// /Chiller_2_Values
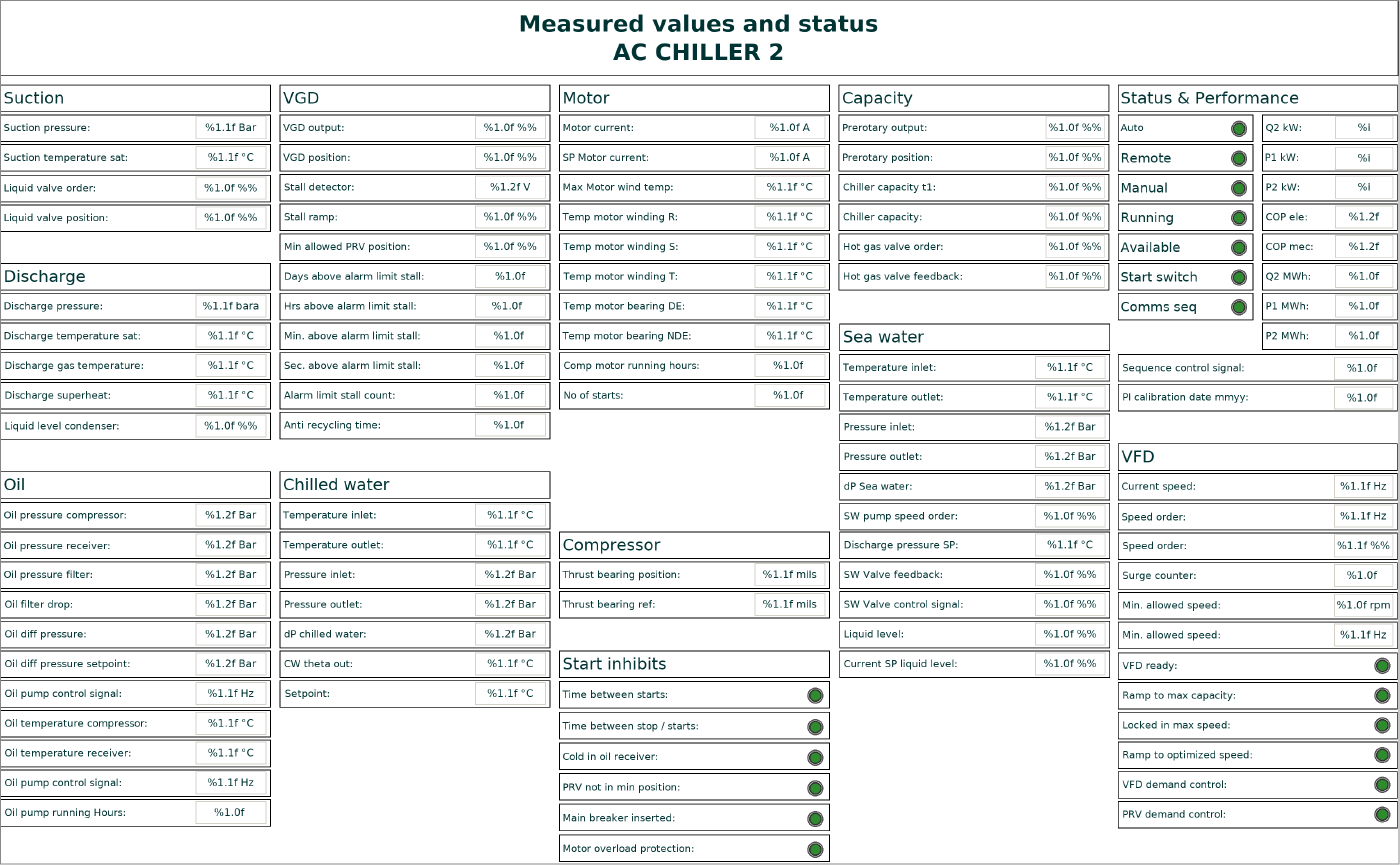
VISUALIZATION Chiller_2_Values  // 1553x960
    Rectangle (0,0 1551x84)
    Label (319,7 912x70), "Measured values and status AC CHILLER 2"
    Rectangle (0,94 300x30)
    Label (1,94 215x30), "Suction"
    Rectangle (0,127 300x30)
    Label (1,122 208x40), "Suction pressure:"
    Textfield (217,129 78x25), "%1.1f Bar", tooltip "Chiller_2.Press_suction_compr", text variable: Chiller_2.Press_suction_compr
        p4168582468: Chiller_2.Press_suction_compr
    Rectangle (0,160 300x30)
    Label (1,155 209x40), "Suction temperature sat:"
    Textfield (217,162 78x25), "%1.1f °C", tooltip "Chiller_2.Suction_saturated_temp", text variable: Chiller_2.Suction_saturated_temp
        p4168582468: Chiller_2.Suction_saturated_temp
    Rectangle (0,194 300x30)
    Label (1,189 211x40), "Liquid valve order:"
    Textfield (217,196 78x25), "%1.0f %%", tooltip "Chiller_2.Liquid_valve_output", text variable: Chiller_2.Liquid_valve_output
        p4168582468: Chiller_2.Liquid_valve_output
    Rectangle (0,227 300x30)
    Label (1,222 216x40), "Liquid valve position:"
    Textfield (217,229 78x25), "%1.0f %%", tooltip "Chiller_2.Feedback_liquid_valve", text variable: Chiller_2.Feedback_liquid_valve
        p4168582468: Chiller_2.Feedback_liquid_valve
    Rectangle (310,94 300x30)
    Label (311,94 194x30), "VGD"
    Rectangle (310,127 300x30)
    Label (311,122 209x40), "VGD output:"
    Textfield (527,129 78x25), "%1.0f %%", tooltip "Chiller_2.VGD_output", text variable: Chiller_2.VGD_output
        p4168582468: Chiller_2.VGD_output
    Rectangle (310,160 300x30)
    Label (311,155 204x40), "VGD position:"
    Textfield (527,162 78x25), "%1.0f %%", tooltip "Chiller_2.Feedback_VGD", text variable: Chiller_2.Feedback_VGD
        p4168582468: Chiller_2.Feedback_VGD
    Rectangle (310,193 300x30)
    Label (312,188 209x40), "Stall detector:"
    Textfield (527,195 78x25), "%1.2f V", tooltip "Chiller_2.Stall_detector", text variable: Chiller_2.Stall_detector
        p4168582468: Chiller_2.Stall_detector
    Rectangle (310,226 300x30)
    Label (312,221 178x40), "Stall ramp:"
    Textfield (527,228 78x25), "%1.0f %%", tooltip "Chiller_2.Stall_ramp", text variable: Chiller_2.Stall_ramp
        p4168582468: Chiller_2.Stall_ramp
    Rectangle (310,259 300x30)
    Label (312,254 216x40), "Min allowed PRV position:"
    Textfield (527,261 78x25), "%1.0f %%", tooltip "Chiller_2.Min_allowed_PRVposition", text variable: Chiller_2.Min_allowed_PRVposition
        p4168582468: Chiller_2.Min_allowed_PRVposition
    Rectangle (310,292 300x30)
    Label (312,287 216x40), "Days above alarm limit stall:"
    Textfield (527,294 78x25), "%1.0f", tooltip "Chiller_2.Days_above_stall_limit", text variable: Chiller_2.Days_above_stall_limit
        p4168582468: Chiller_2.Days_above_stall_limit
    Rectangle (310,325 300x30)
    Label (312,320 215x40), "Hrs above alarm limit stall:"
    Textfield (527,327 78x25), "%1.0f", tooltip "Chiller_2.Hrs_above_stall_limit", text variable: Chiller_2.Hrs_above_stall_limit
        p4168582468: Chiller_2.Hrs_above_stall_limit
    Rectangle (310,358 300x30)
    Label (312,353 218x40), "Min. above alarm limit stall:"
    Textfield (527,360 78x25), "%1.0f", tooltip "Chiller_2.Min_above_stall_limit", text variable: Chiller_2.Min_above_stall_limit
        p4168582468: Chiller_2.Min_above_stall_limit
    Rectangle (310,391 300x30)
    Label (312,386 214x40), "Sec. above alarm limit stall:"
    Textfield (527,393 78x25), "%1.0f", tooltip "Chiller_2.Sec_above_stall_limit", text variable: Chiller_2.Sec_above_stall_limit
        p4168582468: Chiller_2.Sec_above_stall_limit
    Rectangle (310,424 300x30)
    Label (312,419 216x40), "Alarm limit stall count:"
    Textfield (527,426 78x25), "%1.0f", tooltip "Chiller_2.Alarm_limit_stall_count", text variable: Chiller_2.Alarm_limit_stall_count
        p4168582468: Chiller_2.Alarm_limit_stall_count
    Rectangle (930,94 300x30)
    Label (931,94 162x30), "Capacity"
    Rectangle (930,127 300x30)
    Label (931,126 174x32), "Prerotary output:"
    Textfield (1160,129 65x25), "%1.0f %%", tooltip "Chiller_2.Prerotary_output", text variable: Chiller_2.Prerotary_output
        p4168582468: Chiller_2.Prerotary_output
    Rectangle (930,160 300x30)
    Label (931,159 173x32), "Prerotary position:"
    Textfield (1160,162 65x25), "%1.0f %%", tooltip "Chiller_2.Feedback_PRV", text variable: Chiller_2.Feedback_PRV
        p4168582468: Chiller_2.Feedback_PRV
    Rectangle (930,259 300x30)
    Label (932,258 177x32), "Hot gas valve order:"
    Textfield (1160,261 65x25), "%1.0f %%", tooltip "Chiller_2.Hot_gas_valve_output", text variable: Chiller_2.Hot_gas_valve_output
        p4168582468: Chiller_2.Hot_gas_valve_output
    Rectangle (930,292 300x30)
    Label (932,293 177x28), "Hot gas valve feedback:"
    Textfield (1160,294 65x25), "%1.0f %%", tooltip "Chiller_2.Feedback_HGV", text variable: Chiller_2.Feedback_HGV
        p4168582468: Chiller_2.Feedback_HGV
    Rectangle (0,292 300x30)
    Label (1,292 194x30), "Discharge"
    Rectangle (0,325 300x30)
    Label (1,320 213x40), "Discharge pressure:"
    Textfield (217,327 78x25), "%1.1f bara", tooltip "Chiller_2.Press_discharge_compr", text variable: Chiller_2.Press_discharge_compr
        p4168582468: Chiller_2.Press_discharge_compr
    Rectangle (0,358 300x30)
    Label (1,353 214x40), "Discharge temperature sat:"
    Textfield (217,360 78x25), "%1.1f °C", tooltip "Chiller_2.Discharge_saturated_temp", text variable: Chiller_2.Discharge_saturated_temp
        p4168582468: Chiller_2.Discharge_saturated_temp
    Rectangle (0,391 300x30)
    Label (2,386 213x40), "Discharge gas temperature:"
    Textfield (217,393 78x25), "%1.1f °C", tooltip "Chiller_2.Temp_discharge", text variable: Chiller_2.Temp_discharge
        p4168582468: Chiller_2.Temp_discharge
    Rectangle (0,458 300x30)
    Textfield (217,460 78x25), "%1.0f %%", tooltip "Chiller_2.Liquid_level_condenser", text variable: Chiller_2.Liquid_level_condenser
        p4168582468: Chiller_2.Liquid_level_condenser
    Rectangle (0,424 300x30)
    Label (2,419 212x40), "Discharge superheat:"
    Textfield (217,426 78x25), "%1.1f °C", tooltip "Chiller_2.Discharge_superheat", text variable: Chiller_2.Discharge_superheat
        p4168582468: Chiller_2.Discharge_superheat
    Label (2,453 210x40), "Liquid level condenser:"
    Rectangle (1240,127 150x30)
    Rectangle (1240,160 150x30)
    Rectangle (1240,193 150x30)
    Rectangle (1240,226 150x30)
    Rectangle (1240,259 150x30)
    Rectangle (1240,292 150x30)
    Rectangle (1240,325 150x30)
    Lamp1 (1363,133 23x20), tooltip "Chiller_2.Unit_auto", variable: Chiller_2.Unit_auto, style: Lamp-Lamp1-Green
    Label (1240,129 112x26), "Auto"
    Label (1240,165 105x21), "Remote"
    Lamp1 (1363,166 23x20), tooltip "Chiller_2.Unit_remote", variable: Chiller_2.Unit_remote, style: Lamp-Lamp1-Green
    Label (1240,198 105x21), "Manual"
    Lamp1 (1363,199 23x20), tooltip "Chiller_2.Unit_manual", variable: Chiller_2.Unit_manual, style: Lamp-Lamp1-Green
    Label (1240,231 105x21), "Running"
    Lamp1 (1363,232 23x20), tooltip "Chiller_2.Unit_running", variable: Chiller_2.Unit_running, style: Lamp-Lamp1-Green
    Label (1240,264 105x21), "Available"
    Lamp1 (1363,265 23x20), tooltip "Chiller_2.Unit_avabiable", variable: Chiller_2.Unit_available, style: Lamp-Lamp1-Green
    Label (1240,297 104x21), "Start switch"
    Lamp1 (1363,298 23x20), tooltip "Chiller_2.Unit_start_switch", variable: Chiller_2.Unit_start_switch, style: Lamp-Lamp1-Green
    Lamp1 (1363,331 23x20), tooltip "Sequence.A_Comms_Chiller_2", variable: not.Sequence.A_Comms_Chiller_2, style: Lamp-Lamp1-Green
    Label (1240,330 107x21), "Comms seq"
    Rectangle (930,193 300x30)
    Label (932,192 174x32), "Chiller capacity t1:"
    Textfield (1160,195 65x25), "%1.0f %%", tooltip "Chiller_2.Chiller_capacity_t1", text variable: Chiller_2.Chiller_capacity_t1
        p4168582468: Chiller_2.Chiller_capacity_t1
    Rectangle (620,94 300x30)
    Label (621,94 194x30), "Motor"
    Rectangle (620,127 300x30)
    Label (621,122 209x40), "Motor current:"
    Textfield (837,129 78x25), "%1.0f A", tooltip "Chiller_2.Motor_current", text variable: Chiller_2.Motor_current
        p4168582468: Chiller_2.Motor_current
    Rectangle (620,226 300x30)
    Label (621,221 210x40), "Temp motor winding R:"
    Textfield (837,228 78x25), "%1.1f °C", tooltip "Chiller_2.Temp_motor_wind_R", text variable: Chiller_2.Temp_motor_wind_R
        p4168582468: Chiller_2.Temp_motor_wind_R
    Rectangle (620,259 300x30)
    Label (622,254 204x40), "Temp motor winding S:"
    Textfield (837,261 78x25), "%1.1f °C", tooltip "Chiller_2.Temp_motor_wind_S", text variable: Chiller_2.Temp_motor_wind_S
        p4168582468: Chiller_2.Temp_motor_wind_S
    Rectangle (620,292 300x30)
    Label (622,287 206x40), "Temp motor winding T:"
    Textfield (837,294 78x25), "%1.1f °C", tooltip "Chiller_2.Temp_motor_wind_T", text variable: Chiller_2.Temp_motor_wind_T
        p4168582468: Chiller_2.Temp_motor_wind_T
    Rectangle (620,325 300x30)
    Label (622,320 216x40), "Temp motor bearing DE:"
    Textfield (837,327 78x25), "%1.1f °C", tooltip "Chiller_2.Temp_motor_bearing_DE", text variable: Chiller_2.Temp_motor_bearing_DE
        p4168582468: Chiller_2.Temp_motor_bearing_DE
    Rectangle (620,358 300x30)
    Label (621,353 218x40), "Temp motor bearing NDE:"
    Textfield (837,360 78x25), "%1.1f °C", tooltip "Chiller_2.Temp_motor_bearing_NDE", text variable: Chiller_2.Temp_motor_bearing_NDE
        p4168582468: Chiller_2.Temp_motor_bearing_NDE
    Rectangle (620,391 300x30)
    Label (622,386 214x40), "Comp motor running hours:"
    Textfield (837,393 78x25), "%1.0f", tooltip "Chiller_2.Running_hours_compressormotor", text variable: Chiller_2.Running_hours_compressormotor
        p4168582468: Chiller_2.Running_hours_compressormotor
    Rectangle (620,424 300x30)
    Label (622,419 207x40), "No of starts:"
    Textfield (837,426 78x25), "%1.0f", tooltip "Chiller_2.Number_of_starts", text variable: Chiller_2.Number_of_starts
        p4168582468: Chiller_2.Number_of_starts
    Rectangle (310,523 300x30)
    Label (311,523 194x30), "Chilled water"
    Rectangle (310,557 300x30)
    Label (311,552 204x40), "Temperature inlet:"
    Textfield (527,559 78x25), "%1.1f °C", tooltip "Chiller_2.Temp_chilled_medium_in", text variable: Chiller_2.Temp_chilled_medium_in
        p4168582468: Chiller_2.Temp_chilled_medium_in
    Rectangle (310,590 300x30)
    Label (311,585 209x40), "Temperature outlet:"
    Textfield (527,592 78x25), "%1.1f °C", tooltip "Chiller_2.Temp_chilled_medium_out", text variable: Chiller_2.Temp_chilled_medium_out
        p4168582468: Chiller_2.Temp_chilled_medium_out
    Rectangle (310,623 300x30)
    Label (312,618 206x40), "Pressure inlet:"
    Textfield (527,625 78x25), "%1.2f Bar", tooltip "Chiller_2.Press_chilled_medium_in", text variable: Chiller_2.Press_chilled_medium_in
        p4168582468: Chiller_2.Press_chilled_medium_in
    Rectangle (310,656 300x30)
    Label (312,651 208x40), "Pressure outlet:"
    Textfield (527,658 78x25), "%1.2f Bar", tooltip "Chiller_2.Press_chilled_medium_out", text variable: Chiller_2.Press_chilled_medium_out
        p4168582468: Chiller_2.Press_chilled_medium_out
    Rectangle (310,689 300x30)
    Label (312,684 207x40), "dP chilled water:"
    Textfield (527,691 78x25), "%1.2f Bar", tooltip "Chiller_2.dP_CW", text variable: Chiller_2.dP_CW
        p4168582468: Chiller_2.dP_CW
    Rectangle (310,722 300x30)
    Label (312,717 205x40), "CW theta out:"
    Textfield (527,724 78x25), "%1.1f °C", tooltip "Chiller_2.Theta_out", text variable: Chiller_2.Theta_out
        p4168582468: Chiller_2.Theta_out
    Rectangle (310,755 300x30)
    Label (313,750 205x40), "Setpoint:"
    Textfield (527,757 78x25), "%1.1f °C", tooltip "Chiller_2.SP_CW_controller", text variable: Chiller_2.SP_CW_controller
        p4168582468: Chiller_2.SP_CW_controller
    Rectangle (620,160 300x30)
    Label (621,155 209x40), "SP Motor current:"
    Textfield (837,162 78x25), "%1.0f A", tooltip "Chiller_2.SP_MC_controller", text variable: Chiller_2.SP_MC_controller
        p4168582468: Chiller_2.SP_MC_controller
    Rectangle (620,590 300x30)
    Label (621,590 194x30), "Compressor"
    Rectangle (620,623 300x30)
    Label (621,622 216x32), "Thrust bearing position:"
    Textfield (837,625 78x25), "%1.1f mils", tooltip "Chiller_2.Thrust_bearing_position", text variable: Chiller_2.Thrust_bearing_position
        p4168582468: Chiller_2.Thrust_bearing_position
    Rectangle (620,656 300x30)
    Label (621,655 216x32), "Thrust bearing ref:"
    Textfield (837,658 78x25), "%1.1f mils", tooltip "Chiller_2.Thrust_bearing_ref", text variable: Chiller_2.Thrust_bearing_ref
        p4168582468: Chiller_2.Thrust_bearing_ref
    Rectangle (310,457 300x30)
    Label (312,452 216x40), "Anti recycling time:"
    Textfield (527,459 78x25), "%1.0f", tooltip "Chiller_2.Anti_recycle_time", text variable: Chiller_2.Anti_recycle_time
        p4168582468: Chiller_2.Anti_recycle_time
    Rectangle (0,523 300x30)
    Label (1,523 194x30), "Oil"
    Rectangle (0,557 300x30)
    Label (1,552 211x40), "Oil pressure compressor:"
    Textfield (217,559 78x25), "%1.2f Bar", tooltip "Chiller_2.Press_oil_compr", text variable: Chiller_2.Press_oil_compr
        p4168582468: Chiller_2.Press_oil_compr
    Rectangle (0,590 300x30)
    Label (1,586 210x40), "Oil pressure receiver:"
    Textfield (217,592 78x25), "%1.2f Bar", tooltip "Chiller_2.Press_oil_receiver", text variable: Chiller_2.Press_oil_receiver
        p4168582468: Chiller_2.Press_oil_receiver
    Rectangle (0,656 300x30)
    Label (2,651 209x40), "Oil filter drop:"
    Textfield (217,658 78x25), "%1.2f Bar", tooltip "Chiller_2.Oil_Filter_Drop", text variable: Chiller_2.Oil_Filter_Drop
        p4168582468: Chiller_2.Oil_Filter_Drop
    Rectangle (0,689 300x30)
    Label (2,684 211x40), "Oil diff pressure:"
    Textfield (217,691 78x25), "%1.2f Bar", tooltip "Chiller_2.Oil_diff_pressure", text variable: Chiller_2.Oil_diff_pressure
        p4168582468: Chiller_2.Oil_diff_pressure
    Rectangle (0,788 300x30)
    Label (2,791 218x24), "Oil temperature compressor:"
    Textfield (217,790 78x25), "%1.1f °C", tooltip "Chiller_2.Temp_oil_inlet_compr", text variable: Chiller_2.Temp_oil_inlet_compr
        p4168582468: Chiller_2.Temp_oil_inlet_compr
    Rectangle (0,821 300x30)
    Label (2,816 210x40), "Oil temperature receiver:"
    Textfield (217,823 78x25), "%1.1f °C", tooltip "Chiller_2.Oil_temp_receiver", text variable: Chiller_2.Oil_temp_receiver
        p4168582468: Chiller_2.Oil_temp_receiver
    Rectangle (0,854 300x30)
    Label (2,849 212x40), "Oil pump control signal:"
    Textfield (217,856 78x25), "%1.1f Hz", tooltip "Chiller_2.Setpoint_conv_oil_pump", text variable: Chiller_2.Setpoint_conv_oil_pump
        p4168582468: Chiller_2.Setpoint_conv_oil_pump
    Rectangle (0,887 300x30)
    Label (2,882 206x40), "Oil pump running Hours:"
    Textfield (217,889 78x25), "%1.0f", tooltip "Chiller_2.Oil_pump_running_hours", text variable: Chiller_2.Oil_pump_running_hours
        p4168582468: Chiller_2.Oil_pump_running_hours
    Rectangle (0,623 300x30)
    Label (1,618 210x40), "Oil pressure filter:"
    Textfield (217,625 78x25), "%1.2f Bar", tooltip "Chiller_2.Oil_pressure_before_filter", text variable: Chiller_2.Oil_pressure_before_filter
        p4168582468: Chiller_2.Oil_pressure_before_filter
    Rectangle (0,722 300x30)
    Label (2,724 211x26), "Oil diff pressure setpoint:"
    Textfield (217,724 78x25), "%1.2f Bar", tooltip "Chiller_2.SP_oil_pressure", text variable: Chiller_2.SP_oil_pressure
        p4168582468: Chiller_2.SP_oil_pressure
    Rectangle (620,193 300x30)
    Label (621,188 210x40), "Max Motor wind temp:"
    Textfield (837,195 78x25), "%1.1f °C", tooltip "Chiller_2.Max_motor_wind_temp", text variable: Chiller_2.Max_motor_wind_temp
        p4168582468: Chiller_2.Max_motor_wind_temp
    Rectangle (931,359 300x30)
    Label (932,359 194x30), "Sea water"
    Rectangle (931,393 300x30)
    Label (932,388 211x40), "Temperature inlet:"
    Textfield (1148,395 78x25), "%1.1f °C", tooltip "Chiller_2.Temp_water_inlet_cond", text variable: Chiller_2.Temp_water_inlet_cond
        p4168582468: Chiller_2.Temp_water_inlet_cond
    Rectangle (931,459 300x30)
    Label (933,454 210x40), "Pressure inlet:"
    Textfield (1148,461 78x25), "%1.2f Bar", tooltip "Chiller_2.Press_water_cond_inlet", text variable: Chiller_2.Press_water_cond_inlet
        p4168582468: Chiller_2.Press_water_cond_inlet
    Rectangle (931,492 300x30)
    Label (933,487 210x40), "Pressure outlet:"
    Textfield (1148,494 78x25), "%1.2f Bar", tooltip "Chiller_2.Press_water_cond_out", text variable: Chiller_2.Press_water_cond_out
        p4168582468: Chiller_2.Press_water_cond_out
    Rectangle (931,525 300x30)
    Label (933,520 210x40), "dP Sea water:"
    Textfield (1148,527 78x25), "%1.2f Bar", tooltip "Chiller_2.dP_CW", text variable: Chiller_2.dP_SW
        p4168582468: Chiller_2.dP_SW
    Rectangle (931,558 300x30)
    Label (933,553 216x40), "SW pump speed order:"
    Textfield (1148,560 78x25), "%1.0f %%", tooltip "Chiller_2.SW_pump_speed_order", text variable: Chiller_2.SW_pump_speed_order
        p4168582468: Chiller_2.SW_pump_speed_order
    Rectangle (931,426 300x30)
    Label (932,421 211x40), "Temperature outlet:"
    Textfield (1148,428 78x25), "%1.1f °C", tooltip "Chiller_2.Temp_water_outlet_cond", text variable: Chiller_2.Temp_water_outlet_cond
        p4168582468: Chiller_2.Temp_water_outlet_cond
    Rectangle (931,590 300x30)
    Label (933,585 208x40), "Discharge pressure SP:"
    Textfield (1148,592 78x25), "%1.1f °C", tooltip "Chiller_2.SP_cond_press", text variable: Chiller_2.SP_cond_press
        p4168582468: Chiller_2.SP_cond_press
    Rectangle (931,623 300x30)
    Label (933,618 208x40), "SW Valve feedback:"
    Textfield (1148,625 78x25), "%1.0f %%", tooltip "Chiller_2.Feedback_seawater_valve_overboard", text variable: Chiller_2.Feedback_seawater_valve_overboard
        p4168582468: Chiller_2.Feedback_seawater_valve_overboard
    Rectangle (931,656 300x30)
    Label (933,651 208x40), "SW Valve control signal:"
    Textfield (1148,658 78x25), "%1.0f %%", tooltip "Chiller_2.Control_signal_SW_valve", text variable: Chiller_2.Order_SWW_overboard
        p4168582468: Chiller_2.Order_SWW_overboard
    Rectangle (931,689 300x30)
    Label (933,684 208x40), "Liquid level:"
    Textfield (1148,691 78x25), "%1.0f %%", tooltip "Chiller_2.Liquid_level_condenser", text variable: Chiller_2.Liquid_level_condenser
        p4168582468: Chiller_2.Liquid_level_condenser
    Rectangle (931,722 300x30)
    Label (933,717 208x40), "Current SP liquid level:"
    Textfield (1148,724 78x25), "%1.0f %%", tooltip "Chiller_2.SP_PID_Level", text variable: Chiller_2.SP_PID_Level
        p4168582468: Chiller_2.SP_PID_Level
    Rectangle (930,226 300x30)
    Label (932,225 174x32), "Chiller capacity:"
    Textfield (1160,228 65x25), "%1.0f %%", tooltip "Chiller_2.Chiller_capacity", text variable: Chiller_2.Chiller_capacity
        p4168582468: Chiller_2.Chiller_capacity
    Rectangle (1240,393 310x30)
    Label (1242,399 227x19), "Sequence control signal:"
    Textfield (1480,396 65x25), "%1.0f", tooltip "Chiller_2.Control_signal_unit_d", text variable: Chiller_2.Control_signal_unit_d
        p4168582468: Chiller_2.Control_signal_unit_d
    Rectangle (1240,426 310x30)
    Label (1242,429 227x24), "PI calibration date mmyy:"
    Textfield (1480,429 65x25), "%1.0f", tooltip "Chiller_2.Cal_date_MMYY", text variable: Chiller_2.Cal_date_MMYY
        p4168582468: Chiller_2.Cal_date_MMYY
    Rectangle (1400,226 150x30)
    Rectangle (1400,127 150x30)
    Rectangle (1400,193 150x30)
    Rectangle (1400,160 150x30)
    Rectangle (1400,292 150x30)
    Rectangle (1400,259 150x30)
    Rectangle (1400,358 150x30)
    Rectangle (1400,325 150x30)
    Label (1401,228 112x26), "COP ele:"
    Rectangle (1240,94 310x30)
    Label (1240,94 252x30), "Status & Performance"
    Label (1401,126 112x32), "Q2 kW:"
    Label (1401,194 112x28), "P2 kW:"
    Label (1400,159 112x32), "P1 kW:"
    Label (1401,293 112x28), "Q2 MWh:"
    Label (1401,261 112x26), "COP mec:"
    Label (1401,360 112x26), "P2 MWh:"
    Label (1401,327 112x26), "P1 MWh:"
    Textfield (1481,228 64x25), "%1.2f", tooltip "Chiller_2.COP_chiller_ele", text variable: Chiller_2.COP_chiller_ele
        p4168582468: Chiller_2.COP_chiller_ele
    Textfield (1481,129 64x25), "%i", tooltip "Chiller_2.Chiller_capacity_kW", text variable: Chiller_2.Chiller_capacity_kW
        p4168582468: Chiller_2.Chiller_capacity_kW
    Textfield (1481,195 64x25), "%i", tooltip "Chiller_2.P2_mot_1_kW", text variable: Chiller_2.P2_mot_1_kW
        p4168582468: Chiller_2.P2_mot_1_kW
    Textfield (1481,163 64x25), "%i", tooltip "Chiller_2.P1_motor_kW", text variable: Chiller_2.P1_motor_kW
        p4168582468: Chiller_2.P1_motor_kW
    Textfield (1481,294 64x25), "%1.0f", tooltip "Chiller_2.Q2_chillerMWh", text variable: Chiller_2.Q2_chillerMWh
        p4168582468: Chiller_2.Q2_chillerMWh
    Textfield (1481,261 64x25), "%1.2f", tooltip "Chiller_2.COP_chiller_mech", text variable: Chiller_2.COP_chiller_mech
        p4168582468: Chiller_2.COP_chiller_mech
    Textfield (1481,360 64x25), "%1.0f", tooltip "Chiller_2.Chiller_P2_MWh", text variable: Chiller_2.Chiller_P2_MWh
        p4168582468: Chiller_2.Chiller_P2_MWh
    Textfield (1481,327 64x25), "%1.0f", tooltip "Chiller_2.Chiller_P1_MWh", text variable: Chiller_2.Chiller_P1_MWh
        p4168582468: Chiller_2.Chiller_P1_MWh
    Rectangle (0,755 300x30)
    Label (2,757 211x26), "Oil pump control signal:"
    Textfield (217,757 78x25), "%1.1f Hz", tooltip "Chiller_2.Setpoint_conv_oil_pump", text variable: Chiller_2.Setpoint_conv_oil_pump
        p4168582468: Chiller_2.Setpoint_conv_oil_pump
    Rectangle (620,722 300x30)
    Label (621,722 194x30), "Start inhibits"
    Rectangle (620,756 300x30)
    Label (621,755 216x32), "Time between starts:"
    Rectangle (620,790 300x30)
    Label (621,790 216x32), "Time between stop / starts:"
    Rectangle (620,824 300x30)
    Label (621,824 216x32), "Cold in oil receiver:"
    Rectangle (620,858 300x30)
    Label (621,858 216x32), "PRV not in min position:"
    Rectangle (620,892 300x30)
    Label (621,892 216x32), "Main breaker inserted:"
    Lamp1 (893,762 23x20), variable: Chiller_2.Start_inhib_time_between_Start, style: Lamp-Lamp1-Green
    Lamp1 (893,797 23x20), variable: Chiller_2.Start_inhib_time_between_Stop_Start, style: Lamp-Lamp1-Green
    Lamp1 (893,831 23x20), variable: Chiller_2.Start_inhib_time_Oil_receiver_temp, style: Lamp-Lamp1-Green
    Lamp1 (893,865 23x20), variable: Chiller_2.Start_inhib_PRV_not_min, style: Lamp-Lamp1-Green
    Lamp1 (893,899 23x20), variable: not.Chiller_2.DO_9_0_Main_breaker_ready, style: Lamp-Lamp1-Green
    Rectangle (620,926 300x30)
    Label (621,926 216x32), "Motor overload protection:"
    Lamp1 (893,933 23x20), variable: not.Chiller_2.DI_0_6_Overload_protection, style: Lamp-Lamp1-Green
    Rectangle (1240,492 310x30)
    Rectangle (1240,525 310x30)
    Rectangle (1240,558 310x30)
    Rectangle (1240,591 310x30)
    Rectangle (1240,624 310x30)
    Rectangle (1240,657 310x30)
    Rectangle (1240,690 310x30)
    Rectangle (1240,724 310x30)
    Rectangle (1240,757 310x30)
    Rectangle (1240,790 310x30)
    Rectangle (1240,823 310x30)
    Rectangle (1240,856 310x30)
    Rectangle (1240,889 310x30)
    Label (1241,492 162x30), "VFD"
    Label (1241,524 173x32), "Current speed:"
    Textfield (1480,527 65x25), "%1.1f Hz", tooltip "Chiller_2.Speed_feedback_VFD", text variable: Chiller_2.Speed_feedback_VFD
        p4168582468: Chiller_2.Speed_feedback_VFD
    Label (1241,554 167x40), "Speed order:"
    Textfield (1480,560 65x25), "%1.1f Hz", tooltip "Chiller_2.Order_VFD_Hz", text variable: Chiller_2.Order_VFD_Hz
        p4168582468: Chiller_2.Order_VFD_Hz
    Label (1242,589 171x34), "Speed order:"
    Textfield (1480,593 65x25), "%1.1f %%", tooltip "Chiller_2.Opt_speed_VFD_perc", text variable: Chiller_2.Opt_speed_VFD_perc
        p4168582468: Chiller_2.Opt_speed_VFD_perc
    Label (1242,626 170x26), "Surge counter:"
    Textfield (1480,626 65x25), "%1.0f", tooltip "Chiller_2.Surge_counter_VFD", text variable: Chiller_2.Surge_counter_VFD
        p4168582468: Chiller_2.Surge_counter_VFD
    Label (1242,656 176x32), "Min. allowed speed:"
    Textfield (1480,659 65x25), "%1.0f rpm", tooltip "Chiller_2.VFD_min_allowed_speed", text variable: Chiller_2.VFD_min_allowed_speed
        p4168582468: Chiller_2.VFD_min_allowed_speed
    Label (1242,688 177x34), "Min. allowed speed:"
    Textfield (1480,692 65x25), "%1.1f Hz", tooltip "Chiller_2.VFD_min_allowed_frequence", text variable: Chiller_2.VFD_min_allowed_frequence
        p4168582468: Chiller_2.VFD_min_allowed_frequence
    Label (1242,722 177x34), "VFD ready:"
    Lamp1 (1522,729 23x20), tooltip "Chiller_2.VFD_ready", variable: Chiller_2.VFD_ready, style: Lamp-Lamp1-Green
    Label (1242,755 209x34), "Ramp to max capacity:"
    Lamp1 (1522,762 23x20), tooltip "Chiller_2.VFD_ramp_100_perc", variable: Chiller_2.VFD_ramp_100_perc, style: Lamp-Lamp1-Green
    Label (1242,788 209x34), "Locked in max speed:"
    Lamp1 (1522,795 23x20), tooltip "Chiller_2.VFD_locked_100_perc", variable: Chiller_2.VFD_locked_100_perc, style: Lamp-Lamp1-Green
    Label (1242,821 209x34), "Ramp to optimized speed:"
    Lamp1 (1522,828 23x20), tooltip "Chiller_2.VFD_ramp_d_PRVcontrol", variable: Chiller_2.VFD_ramp_d_PRVcontrol, style: Lamp-Lamp1-Green
    Label (1242,854 209x34), "VFD demand control:"
    Lamp1 (1522,861 23x20), tooltip "Chiller_2.VFD_control", variable: Chiller_2.VFD_control, style: Lamp-Lamp1-Green
    Label (1242,887 209x34), "PRV demand control:"
    Lamp1 (1522,894 23x20), tooltip "Chiller_2.PRV_control", variable: Chiller_2.PRV_control, style: Lamp-Lamp1-Green
END_VISUALIZATION

// /Chiller_2_VFD
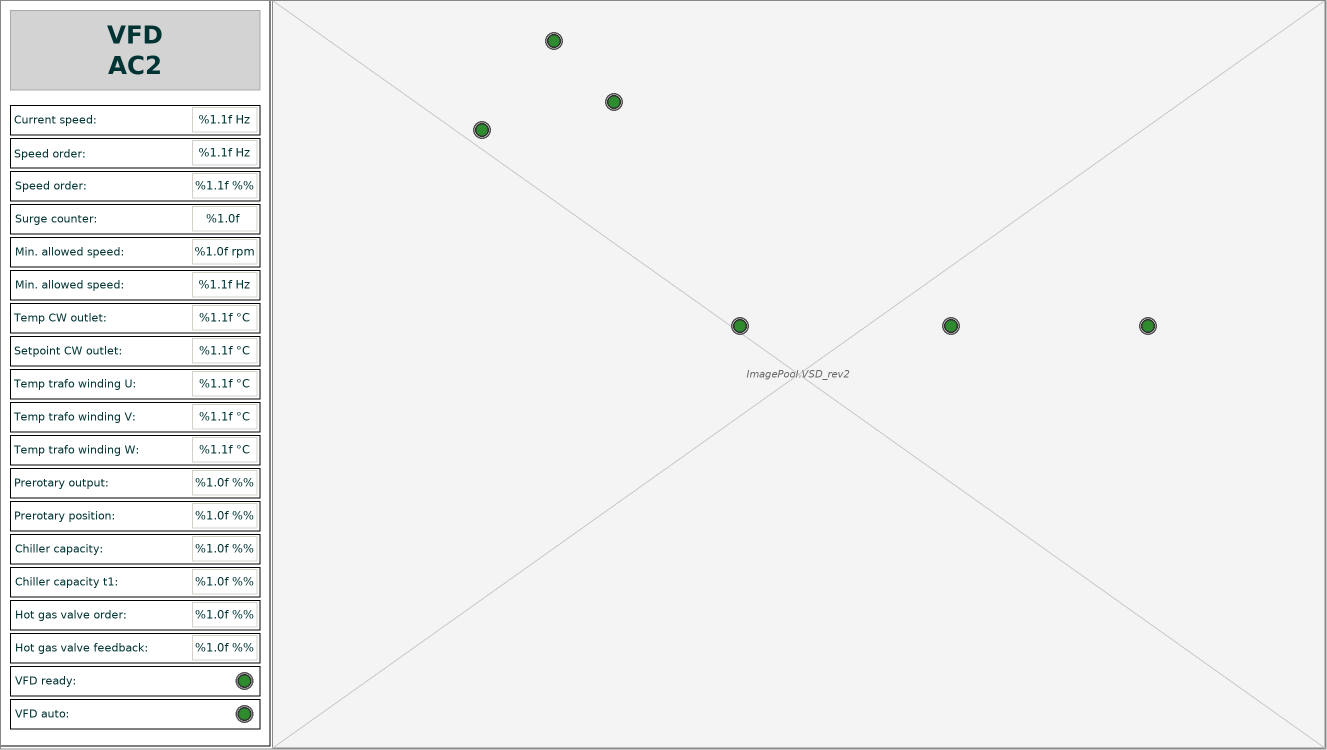
VISUALIZATION Chiller_2_VFD  // 1327x750
    Image (272,0 1053x748), image: ImagePool.VSD_rev2
    Rectangle (0,0 270x746)
    Lamp1 (469,120 26x20), variable: Chiller_2.VFD_ramp_100_perc, style: Lamp-Lamp1-Green
    Lamp1 (541,31 26x20), variable: Chiller_2.VFD_locked_100_perc, style: Lamp-Lamp1-Green
    Lamp1 (601,92 26x20), variable: Chiller_2.VFD_ramp_d_PRVcontrol, style: Lamp-Lamp1-Green
    Lamp1 (727,316 26x20), variable: Chiller_2.PRV_control, style: Lamp-Lamp1-Green
    Lamp1 (938,316 26x20), variable: Chiller_2.VFD_control, style: Lamp-Lamp1-Green
    Lamp1 (1135,316 26x20), variable: Chiller_2.PRV_control, style: Lamp-Lamp1-Green
    Textfield (10,10 250x80), "VFD AC2", text index: Sequence.Seq_cap_order_C3
    Rectangle (10,666 250x30)
    Label (12,664 177x34), "VFD ready:"
    Lamp1 (233,671 23x20), tooltip "Chiller_2.VFD_ready", variable: Chiller_2.VFD_ready, style: Lamp-Lamp1-Green
    Rectangle (10,699 250x30)
    Label (12,697 177x34), "VFD auto:"
    Lamp1 (233,704 23x20), tooltip "Chiller_2.VFD_man_auto", variable: Chiller_2.VFD_man_auto, style: Lamp-Lamp1-Green
    Rectangle (10,105 250x30)
    Label (11,104 173x32), "Current speed:"
    Textfield (192,107 65x25), "%1.1f Hz", tooltip "Chiller_2.Speed_feedback_VFD", text variable: Chiller_2.Speed_feedback_VFD
        p4168582468: Chiller_2.Speed_feedback_VFD
    Rectangle (10,138 250x30)
    Label (11,134 167x40), "Speed order:"
    Textfield (192,140 65x25), "%1.1f Hz", tooltip "Chiller_2.Order_VFD_Hz", text variable: Chiller_2.Order_VFD_Hz
        p4168582468: Chiller_2.Order_VFD_Hz
    Rectangle (10,171 250x30)
    Label (12,169 171x34), "Speed order:"
    Textfield (192,173 65x25), "%1.1f %%", tooltip "Chiller_2.Opt_speed_VFD_perc", text variable: Chiller_2.Opt_speed_VFD_perc
        p4168582468: Chiller_2.Opt_speed_VFD_perc
    Rectangle (10,204 250x30)
    Label (12,206 170x26), "Surge counter:"
    Textfield (192,206 65x25), "%1.0f", tooltip "Chiller_2.Surge_counter_VFD", text variable: Chiller_2.Surge_counter_VFD
        p4168582468: Chiller_2.Surge_counter_VFD
    Rectangle (10,237 250x30)
    Label (12,236 176x32), "Min. allowed speed:"
    Textfield (192,239 65x25), "%1.0f rpm", tooltip "Chiller_2.VFD_min_allowed_speed", text variable: Chiller_2.VFD_min_allowed_speed
        p4168582468: Chiller_2.VFD_min_allowed_speed
    Rectangle (10,270 250x30)
    Label (12,268 177x34), "Min. allowed speed:"
    Textfield (192,272 65x25), "%1.1f Hz", tooltip "Chiller_2.VFD_min_allowed_frequence", text variable: Chiller_2.VFD_min_allowed_frequence
        p4168582468: Chiller_2.VFD_min_allowed_frequence
    Rectangle (10,303 250x30)
    Label (11,305 169x26), "Temp CW outlet:"
    Textfield (192,305 65x25), "%1.1f °C", tooltip "Chiller_2.Temp_chilled_medium_out", text variable: Chiller_2.Temp_chilled_medium_out
        p4168582468: Chiller_2.Temp_chilled_medium_out
    Rectangle (10,336 250x30)
    Label (11,338 169x26), "Setpoint CW outlet:"
    Textfield (192,338 65x25), "%1.1f °C", tooltip "Chiller_2.SP_CW_controller", text variable: Chiller_2.SP_CW_controller
        p4168582468: Chiller_2.SP_CW_controller
    Rectangle (10,369 250x30)
    Label (11,371 169x26), "Temp trafo winding U:"
    Textfield (192,371 65x25), "%1.1f °C", tooltip "Chiller_2.Temp_motor_wind_R", text variable: Chiller_2.Temp_motor_wind_R
        p4168582468: Chiller_2.Temp_motor_wind_R
    Rectangle (10,402 250x30)
    Label (11,404 169x26), "Temp trafo winding V:"
    Textfield (192,404 65x25), "%1.1f °C", tooltip "Chiller_2.Temp_motor_wind_S", text variable: Chiller_2.Temp_motor_wind_S
        p4168582468: Chiller_2.Temp_motor_wind_S
    Rectangle (10,435 250x30)
    Label (11,437 169x26), "Temp trafo winding W:"
    Textfield (192,437 65x25), "%1.1f °C", tooltip "Chiller_2.Temp_motor_wind_T", text variable: Chiller_2.Temp_motor_wind_T
        p4168582468: Chiller_2.Temp_motor_wind_T
    Rectangle (10,468 250x30)
    Label (11,467 174x32), "Prerotary output:"
    Textfield (192,470 65x25), "%1.0f %%", tooltip "Chiller_2.Prerotary_output", text variable: Chiller_2.Prerotary_output
        p4168582468: Chiller_2.Prerotary_output
    Rectangle (10,501 250x30)
    Label (11,500 173x32), "Prerotary position:"
    Textfield (192,503 65x25), "%1.0f %%", tooltip "Chiller_2.Feedback_PRV", text variable: Chiller_2.Feedback_PRV
        p4168582468: Chiller_2.Feedback_PRV
    Rectangle (10,534 250x30)
    Label (12,533 174x32), "Chiller capacity:"
    Textfield (192,536 65x25), "%1.0f %%", tooltip "Chiller_2.Chiller_capacity", text variable: Chiller_2.Chiller_capacity
        p4168582468: Chiller_2.Chiller_capacity
    Rectangle (10,600 250x30)
    Label (12,599 177x32), "Hot gas valve order:"
    Textfield (192,602 65x25), "%1.0f %%", tooltip "Chiller_2.Hot_gas_valve_output", text variable: Chiller_2.Hot_gas_valve_output
        p4168582468: Chiller_2.Hot_gas_valve_output
    Rectangle (10,633 250x30)
    Label (12,634 177x28), "Hot gas valve feedback:"
    Textfield (192,635 65x25), "%1.0f %%", tooltip "Chiller_2.Feedback_HGV", text variable: Chiller_2.Feedback_HGV
        p4168582468: Chiller_2.Feedback_HGV
    Rectangle (10,567 250x30)
    Label (12,566 174x32), "Chiller capacity t1:"
    Textfield (192,569 65x25), "%1.0f %%", tooltip "Chiller_2.Chiller_capacity_t1", text variable: Chiller_2.Chiller_capacity_t1
        p4168582468: Chiller_2.Chiller_capacity_t1
    Rectangle (432,18 87x711), colour toggle: Chiller_2.VFD_ramp_100_perc
    Rectangle (518,18 65x711), colour toggle: Chiller_2.VFD_locked_100_perc
    Rectangle (583,18 57x711), colour toggle: Chiller_2.VFD_ramp_d_PRVcontrol
    Rectangle (641,18 199x711), colour toggle: Chiller_2.PRV_control
    Rectangle (1066,18 162x711), colour toggle: Chiller_2.PRV_control
    Rectangle (841,18 225x711), colour toggle: Chiller_2.VFD_control
END_VISUALIZATION

// /Chiller_3_Alarm
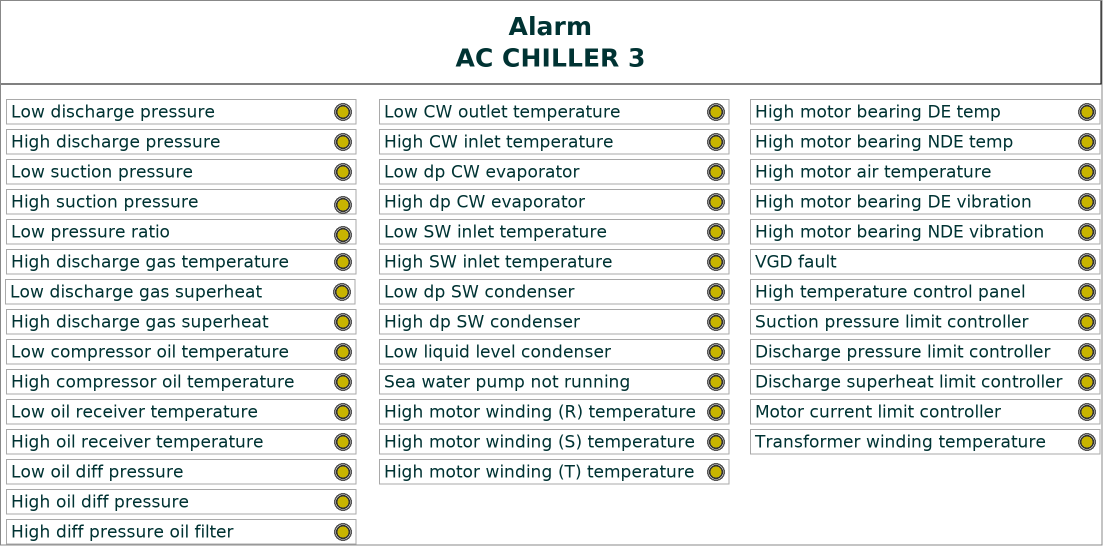
VISUALIZATION Chiller_3_Alarm  // 1103x546
    Rectangle (0,0 1101x84)
    Label (19,7 1063x70), "Alarm AC CHILLER 3"
    Rectangle (750,279 350x25)
    Label (752,281 316x21), "High temperature control panel"
    Lamp1 (1076,282 22x20), variable: Chiller_3.A_High_control_panel_temp, style: Lamp-Lamp1-Yellow
    Rectangle (750,309 350x25)
    Label (752,311 312x21), "Suction pressure limit controller"
    Lamp1 (1076,312 22x20), variable: Chiller_3.A_Suction_press_limit, style: Lamp-Lamp1-Yellow
    Rectangle (6,99 350x25)
    Label (8,101 318x21), "Low discharge pressure"
    Lamp1 (332,102 22x20), variable: Chiller_3.A_low_disch_press, style: Lamp-Lamp1-Yellow
    Rectangle (6,159 350x25)
    Label (8,161 319x21), "Low suction pressure"
    Lamp1 (332,162 22x20), variable: Chiller_3.A_Low_suction_pressure, style: Lamp-Lamp1-Yellow
    Rectangle (6,189 350x25)
    Label (8,191 322x21), "High suction pressure"
    Lamp1 (332,195 22x20), variable: Chiller_3.A_High_suction_pressure, style: Lamp-Lamp1-Yellow
    Rectangle (6,249 350x25)
    Label (8,251 317x21), "High discharge gas temperature"
    Lamp1 (332,252 22x20), variable: Chiller_3.A_High_discharge_temp, style: Lamp-Lamp1-Yellow
    Rectangle (379,399 350x25)
    Label (381,401 320x21), "High motor winding (R) temperature"
    Lamp1 (705,402 22x20), variable: Chiller_3.A_High_motor_wind_temp_R, style: Lamp-Lamp1-Yellow
    Rectangle (379,429 350x25)
    Label (381,431 319x21), "High motor winding (S) temperature"
    Lamp1 (705,432 22x20), variable: Chiller_3.A_High_motor_wind_temp_S, style: Lamp-Lamp1-Yellow
    Rectangle (6,369 350x25)
    Label (8,371 319x21), "High compressor oil temperature"
    Lamp1 (332,372 22x20), variable: Chiller_3.A_High_temp_oil_inlet_comp, style: Lamp-Lamp1-Yellow
    Rectangle (6,339 350x25)
    Label (8,341 322x21), "Low compressor oil temperature"
    Lamp1 (332,342 22x20), variable: Chiller_3.A_Low_temp_oil_inlet_comp, style: Lamp-Lamp1-Yellow
    Rectangle (6,429 350x25)
    Label (8,431 317x21), "High oil receiver temperature"
    Lamp1 (332,432 22x20), variable: Chiller_3.A_High_oil_temp_receiver, style: Lamp-Lamp1-Yellow
    Rectangle (6,399 350x25)
    Label (8,401 319x21), "Low oil receiver temperature"
    Lamp1 (332,402 22x20), variable: Chiller_3.A_Low_oil_temp_receiver, style: Lamp-Lamp1-Yellow
    Rectangle (6,459 350x25)
    Label (8,461 322x21), "Low oil diff pressure"
    Lamp1 (332,462 22x20), variable: Chiller_3.A_Low_oil_diff_pressure, style: Lamp-Lamp1-Yellow
    Rectangle (6,489 350x25)
    Label (8,491 317x21), "High oil diff pressure"
    Lamp1 (332,492 22x20), variable: Chiller_3.A_High_oil_diff_pressure, style: Lamp-Lamp1-Yellow
    Rectangle (6,309 350x25)
    Label (8,311 319x21), "High discharge gas superheat"
    Lamp1 (332,312 22x20), variable: Chiller_3.A_High_discharge_superheat, style: Lamp-Lamp1-Yellow
    Rectangle (5,279 350x25)
    Label (7,281 322x21), "Low discharge gas superheat"
    Lamp1 (331,282 22x20), variable: Chiller_3.A_Low_discharge_superheat, style: Lamp-Lamp1-Yellow
    Rectangle (379,219 350x25)
    Label (381,221 317x21), "Low SW inlet temperature"
    Lamp1 (705,222 22x20), variable: Chiller_3.A_Low_SW_inlet_temp, style: Lamp-Lamp1-Yellow
    Rectangle (379,129 350x25)
    Label (381,131 322x21), "High CW inlet temperature"
    Lamp1 (705,132 22x20), variable: Chiller_3.A_High_CW_inlet_temp, style: Lamp-Lamp1-Yellow
    Rectangle (379,99 350x25)
    Label (381,101 317x21), "Low CW outlet temperature"
    Lamp1 (705,102 22x20), variable: Chiller_3.A_Low_CW_outlet_temp, style: Lamp-Lamp1-Yellow
    Rectangle (6,519 350x25)
    Label (8,521 317x21), "High diff pressure oil filter"
    Lamp1 (332,522 22x20), variable: Chiller_3.A_High_oil_filter_diff_press, style: Lamp-Lamp1-Yellow
    Rectangle (379,459 350x25)
    Label (381,461 317x21), "High motor winding (T) temperature"
    Lamp1 (705,462 22x20), variable: Chiller_3.A_High_motor_wind_temp_T, style: Lamp-Lamp1-Yellow
    Rectangle (750,99 350x25)
    Label (752,101 317x21), "High motor bearing DE temp"
    Lamp1 (1076,102 22x20), variable: Chiller_3.A_High_comp_mo_DE_bear_temp, style: Lamp-Lamp1-Yellow
    Rectangle (750,129 350x25)
    Label (752,131 319x21), "High motor bearing NDE temp"
    Lamp1 (1076,132 22x20), variable: Chiller_3.A_High_comp_mo_NDE_bear_temp, style: Lamp-Lamp1-Yellow
    Rectangle (750,159 350x25)
    Label (752,161 322x21), "High motor air temperature"
    Lamp1 (1076,162 22x20), variable: Chiller_3.A_High_motor_air_temp, style: Lamp-Lamp1-Yellow
    Rectangle (750,189 350x25)
    Label (752,191 317x21), "High motor bearing DE vibration"
    Lamp1 (1076,192 22x20), variable: Chiller_3.A_High_comp_mo_DE_bear_vib, style: Lamp-Lamp1-Yellow
    Rectangle (750,219 350x25)
    Label (752,221 319x21), "High motor bearing NDE vibration"
    Lamp1 (1076,222 22x20), variable: Chiller_3.A_High_comp_mo_NDE_bear_vib, style: Lamp-Lamp1-Yellow
    Rectangle (379,189 350x25)
    Label (381,191 322x21), "High dp CW evaporator"
    Lamp1 (705,192 22x20), variable: Chiller_3.A_High_CW_dP, style: Lamp-Lamp1-Yellow
    Rectangle (379,159 350x25)
    Label (381,161 317x21), "Low dp CW evaporator"
    Lamp1 (705,162 22x20), variable: Chiller_3.A_Low_CW_dP, style: Lamp-Lamp1-Yellow
    Rectangle (379,309 350x25)
    Label (381,311 319x21), "High dp SW condenser"
    Lamp1 (705,312 22x20), variable: Chiller_3.A_High_SW_dP, style: Lamp-Lamp1-Yellow
    Rectangle (379,279 350x25)
    Label (381,281 322x21), "Low dp SW condenser"
    Lamp1 (705,282 22x20), variable: Chiller_3.A_Low_SW_dP, style: Lamp-Lamp1-Yellow
    Rectangle (750,249 350x25)
    Label (752,251 317x21), "VGD fault"
    Lamp1 (1076,252 22x20), variable: Chiller_3.A_VGD_Fault, style: Lamp-Lamp1-Yellow
    Rectangle (379,339 350x25)
    Label (381,341 317x21), "Low liquid level condenser"
    Lamp1 (705,342 22x20), variable: Chiller_3.A_Low_liquid_level, style: Lamp-Lamp1-Yellow
    Rectangle (6,129 350x25)
    Label (8,131 318x21), "High discharge pressure"
    Lamp1 (332,132 22x20), variable: Chiller_3.A_high_disch_press, style: Lamp-Lamp1-Yellow
    Rectangle (379,249 350x25)
    Label (381,251 314x21), "High SW inlet temperature"
    Lamp1 (705,252 22x20), variable: Chiller_3.A_High_SW_inlet_temp, style: Lamp-Lamp1-Yellow
    Rectangle (379,369 350x25)
    Label (381,371 314x21), "Sea water pump not running"
    Lamp1 (705,372 22x20), variable: Chiller_3.A_Seawater_pump_not_running, style: Lamp-Lamp1-Yellow
    Rectangle (750,339 350x25)
    Label (752,341 312x21), "Discharge pressure limit controller"
    Lamp1 (1076,342 22x20), variable: Chiller_3.A_Discharge_press_limit, style: Lamp-Lamp1-Yellow
    Rectangle (750,369 350x25)
    Label (752,371 312x21), "Discharge superheat limit controller"
    Lamp1 (1076,372 22x20), variable: Chiller_3.A_Discharge_superheat_limit, style: Lamp-Lamp1-Yellow
    Rectangle (750,399 350x25)
    Label (752,401 312x21), "Motor current limit controller"
    Lamp1 (1076,402 22x20), variable: Chiller_3.A_Motor_current_limit, style: Lamp-Lamp1-Yellow
    Rectangle (750,429 350x25)
    Label (752,431 312x21), "Transformer winding temperature"
    Lamp1 (1076,432 22x20), variable: Chiller_3.A_Transformer_winding_temp, style: Lamp-Lamp1-Yellow
    Rectangle (6,219 350x25)
    Label (8,221 322x21), "Low pressure ratio"
    Lamp1 (332,225 22x20), variable: Chiller_3.A_Low_press_ratio, style: Lamp-Lamp1-Yellow
END_VISUALIZATION

// /Chiller_3_Flow_Diagram
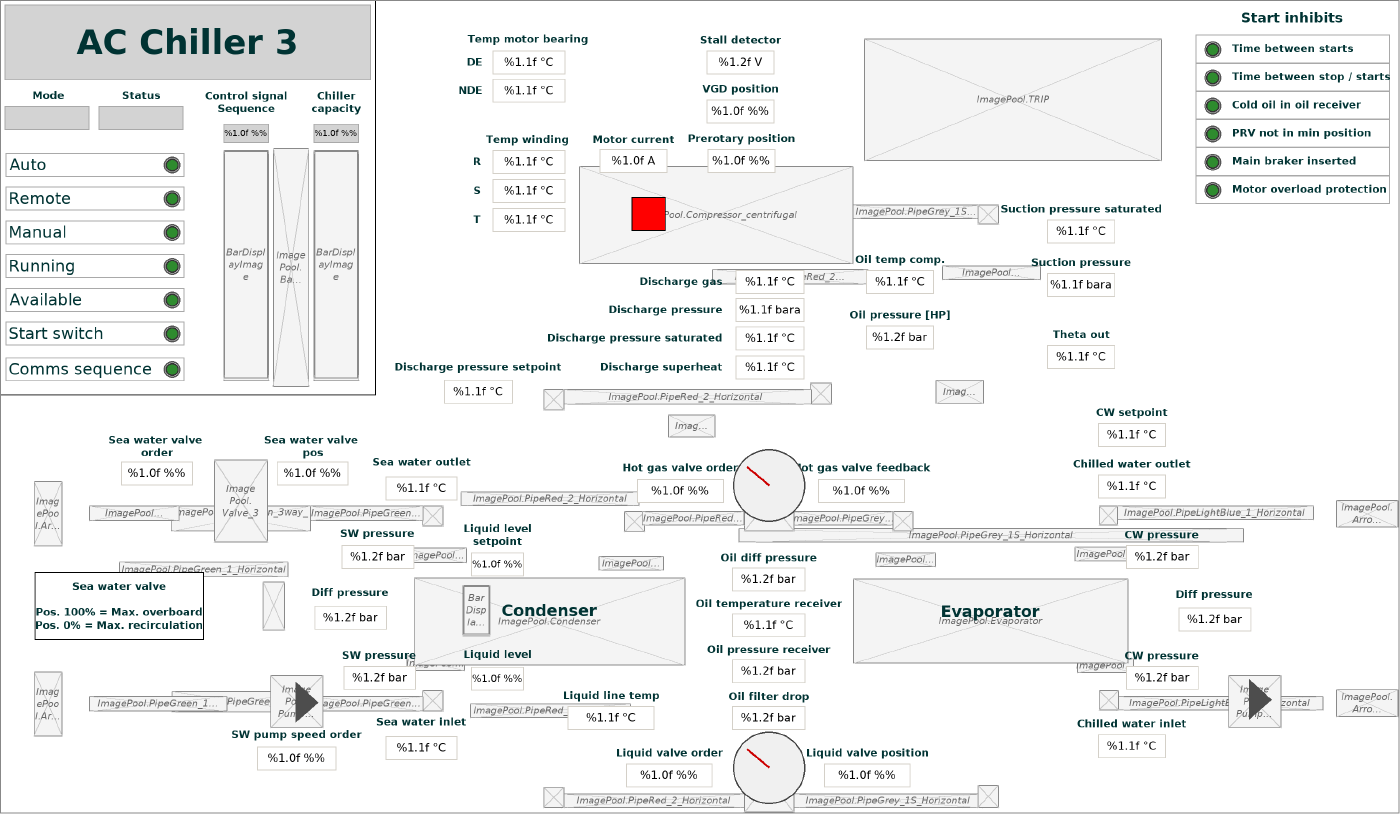
VISUALIZATION Chiller_3_Flow_Diagram  // 1492x868
    Rectangle (0,0 400x421)
    Textfield (238,132 48x20), "%1.0f %%", text variable: Sequence.Seq_cap_order_C3
        p4168582468: Sequence.Seq_cap_order_C3
    Image (1148,702 60x15), angle 270, image: ImagePool.PipeLightBlue_1_Horizontal
    Image (1145,583 67x15), angle 270, image: ImagePool.PipeLightBlue_1_Horizontal
    Image (908,218 137x15), image: ImagePool.PipeGrey_1S_Horizontal
    Image (845,846 202x15), image: ImagePool.PipeGrey_1S_Horizontal
    Image (933,589 64x15), angle 270, image: ImagePool.PipeGrey_1S_Horizontal
    Image (787,563 538x15), angle 270, image: ImagePool.PipeGrey_1S_Horizontal
    Image (843,545 110x15), image: ImagePool.PipeGrey_1S_Horizontal
    Image (638,593 69x15), angle 270, image: ImagePool.PipeRed_2_Horizontal
    Image (501,750 171x15), angle 270, image: ImagePool.PipeRed_2_Horizontal
    Label (218,94 89x30), "Control signal Sequence"
    Image (617,177 292x104), image: ImagePool.Compressor_centrifugal
    Image (759,287 166x16), angle 270, image: ImagePool.PipeRed_2_Horizontal
    Image (863,408 23x23), image: ImagePool.PipeRed_2_LU
    Image (596,415 269x16), image: ImagePool.PipeRed_2_Horizontal
    Image (909,617 293x90), image: ImagePool.Evaporator
    Image (431,584 66x16), angle 270, image: ImagePool.PipeGreen_1_Horizontal
    Image (450,539 22x22), image: ImagePool.PipeGreen_1_LD
    Image (329,539 122x16), image: ImagePool.PipeGreen_1_Horizontal
    Label (331,617 84x30), "Diff pressure"
    Textfield (335,646 77x25), "%1.2f bar", text variable: Chiller_3.dP_SW
        p4168582468: Chiller_3.dP_SW
    Image (127,599 180x16), angle 270, image: ImagePool.PipeGreen_1_Horizontal
    Image (183,737 147x22), image: ImagePool.PipeGreen_3way
    Image (433,699 62x16), angle 270, image: ImagePool.PipeGreen_1_Horizontal
    Image (450,736 22x22), image: ImagePool.PipeGreen_2_LU
    Image (329,742 122x16), image: ImagePool.PipeGreen_1_Horizontal
    Image (182,539 149x27), image: ImagePool.PipeGreen_3way_2
    Image (288,720 56x56), image: ImagePool.Pump_Large_3
    Polygon (315,746) (315,727) (339,749) (315,770) (315,762), colour toggle: Chiller_3.Sea_water_pump
    Image (36,513 30x69), angle 90, image: ImagePool.Arrow green down
    Image (36,716 30x69), angle 270, image: ImagePool.Arrow green down
    Image (579,415 22x22), image: ImagePool.PipeRed_1_RD
    Image (491,524 190x15), angle 270, image: ImagePool.PipeRed_2_Horizontal
    Label (360,554 84x30), "SW pressure"
    Textfield (364,581 77x25), "%1.2f bar", text variable: Chiller_3.Press_water_cond_out
        p4168582468: Chiller_3.Press_water_cond_out
    Image (95,539 96x16), image: ImagePool.PipeGreen_1_Horizontal
    Image (441,616 289x93), image: ImagePool.Condenser
    Image (598,846 197x15), image: ImagePool.PipeRed_2_Horizontal
    Image (579,839 22x22), image: ImagePool.PipeRed_2_RU
    Label (362,684 84x30), "SW pressure"
    Textfield (366,710 77x25), "%1.2f bar", text variable: Chiller_3.Press_water_cond_inlet
        p4168582468: Chiller_3.Press_water_cond_inlet
    Image (793,501 53x65), image: ImagePool.Valve_2
    Image (793,801 53x65), image: ImagePool.Valve_2
    Image (665,545 22x22), image: ImagePool.PipeRed_1_RD
    Image (684,545 109x15), image: ImagePool.PipeRed_2_Horizontal
    Image (951,545 22x21), image: ImagePool.PipeGrey_2_LD
    Image (1042,837 22x24), image: ImagePool.PipeGrey_3_LU
    Image (1042,218 22x21), image: ImagePool.PipeGrey_2_LD
    Image (1004,283 105x15), angle 270, image: ImagePool.PipeGrey_1S_Horizontal
    Label (521,636 129x30), "Condenser"
    Label (991,637 129x30), "Evaporator"
    Image (1189,539 211x15), image: ImagePool.PipeLightBlue_1_Horizontal
    Image (1171,539 20x21), image: ImagePool.PipeLightBlue_3_RD
    Image (1190,742 220x15), image: ImagePool.PipeLightBlue_1_Horizontal
    Image (1171,736 21x21), image: ImagePool.PipeLightBlue_3_RU
    Image (1424,533 66x29), angle 180, image: ImagePool.Arrow lightblue left
    Image (1424,735 66x29), image: ImagePool.Arrow lightblue left
    Image (1309,720 56x56), image: ImagePool.Pump_Large_3
    Polygon (1331,743) (1331,724) (1355,746) (1331,767) (1331,759), colour toggle: Chiller_3.CW_Flow_ind
    Image (280,620 23x52), image: ImagePool.Arrow green down
    Image (712,442 50x24), image: ImagePool.Arrow red left
    Image (997,405 51x25), angle 90, image: ImagePool.Arrow gray left
    Image (291,158 38x254), image: ImagePool.BarScale3
    Label (324,94 69x30), "Chiller capacity"
    Textfield (105,113 90x25), text list: 'TextList_PT', text index: Chiller_3.Unit_switch_status
    Textfield (5,113 90x25), text list: 'TextList_PT', text index: Chiller_3.Unit_start_switch
    Textfield (334,132 48x20), "%1.0f %%", text variable: Chiller_3.Chiller_capacity_t1
        p4168582468: Chiller_3.Chiller_capacity_t1
    Textfield (5,5 390x80), "AC Chiller 3"
    Textfield (525,160 77x25), "%1.1f °C", text variable: Chiller_3.Temp_motor_wind_R
        p4168582468: Chiller_3.Temp_motor_wind_R
    Label (496,160 25x25), "R"
    Textfield (525,191 77x25), "%1.1f °C", text variable: Chiller_3.Temp_motor_wind_S
        p4168582468: Chiller_3.Temp_motor_wind_S
    Label (496,191 25x25), "S"
    Textfield (525,222 77x25), "%1.1f °C", text variable: Chiller_3.Temp_motor_wind_T
        p4168582468: Chiller_3.Temp_motor_wind_T
    Label (496,222 25x25), "T"
    Textfield (679,511 92x25), "%1.0f %%", text variable: Chiller_3.Hot_gas_valve_output
        p4168582468: Chiller_3.Hot_gas_valve_output
    Label (664,484 122x30), "Hot gas valve order"
    Label (849,484 139x30), "Hot gas valve feedback"
    Textfield (872,511 92x25), "%1.0f %%", text variable: Chiller_3.Feedback_HGV
        p4168582468: Chiller_3.Feedback_HGV
    Meter360 (781,479 77x77), value: Chiller_3.Feedback_HGV, style: Meter-Meter360-Gray, scale format: %1.0f, scale 0..100
        p3451962224: ImagePool.Invisible
    Meter360 (781,780 77x77), value: Chiller_3.Feedback_liquid_valve, style: Meter-Meter360-Gray, scale format: %1.0f, scale 0..100
        p3451962224: ImagePool.Invisible
    Textfield (502,589 56x25), "%1.0f %%", text variable: Chiller_3.SP_PID_Level
        p4168582468: Chiller_3.SP_PID_Level
    Label (494,551 73x39), "Liquid level setpoint"
    Textfield (502,711 56x25), "%1.0f %%", text variable: Chiller_3.Liquid_level_condenser
        p4168582468: Chiller_3.Liquid_level_condenser
    Label (491,683 79x30), "Liquid level"
    Textfield (639,159 72x25), "%1.0f A", text variable: Chiller_3.Motor_current
        p4168582468: Chiller_3.Motor_current
    Label (634,138 83x22), "Motor current"
    Textfield (274,796 84x25), "%1.0f %%", text variable: Chiller_3.SW_pump_speed_order
        p4168582468: Chiller_3.SW_pump_speed_order
    Label (250,770 132x27), "SW pump speed order"
    Textfield (473,405 73x25), "%1.1f °C", tooltip "Chiller_3.SP_cond_press", text variable: Chiller_3.SP_cond_press
        p4168582468: Chiller_3.SP_cond_press
    Textfield (784,348 73x25), "%1.1f °C", text variable: Chiller_3.Discharge_saturated_temp
        p4168582468: Chiller_3.Discharge_saturated_temp
    Label (589,347 184x27), "Discharge pressure saturated"
    Label (425,378 169x27), "Discharge pressure setpoint"
    Textfield (411,785 76x25), "%1.1f °C", text variable: Chiller_3.Temp_water_inlet_cond
        p4168582468: Chiller_3.Temp_water_inlet_cond
    Label (399,755 100x30), "Sea water inlet"
    Textfield (411,508 76x25), "%1.1f °C", text variable: Chiller_3.Temp_water_outlet_cond
        p4168582468: Chiller_3.Temp_water_outlet_cond
    Label (397,478 105x30), "Sea water outlet"
    Label (500,27 126x30), "Temp motor bearing"
    Textfield (525,84 77x25), "%1.1f °C", text variable: Chiller_3.Temp_motor_bearing_NDE
        p4168582468: Chiller_3.Temp_motor_bearing_NDE
    Textfield (525,54 77x25), "%1.1f °C", text variable: Chiller_3.Temp_motor_bearing_DE
        p4168582468: Chiller_3.Temp_motor_bearing_DE
    Label (480,54 37x25), "DE"
    Label (480,84 37x25), "NDE"
    Label (678,287 95x27), "Discharge gas"
    Textfield (784,288 73x25), "%1.1f °C", text variable: Chiller_3.Temp_discharge
        p4168582468: Chiller_3.Temp_discharge
    Label (644,317 129x27), "Discharge pressure"
    Textfield (784,318 73x25), "%1.1f bara", text variable: Chiller_3.Press_discharge_compr
        p4168582468: Chiller_3.Press_discharge_compr
    Textfield (784,379 73x25), "%1.1f °C", text variable: Chiller_3.Discharge_superheat
        p4168582468: Chiller_3.Discharge_superheat
    Label (589,378 184x27), "Discharge superheat"
    Label (857,788 135x30), "Liquid valve position"
    Textfield (878,814 92x25), "%1.0f %%", text variable: Chiller_3.Feedback_liquid_valve
        p4168582468: Chiller_3.Feedback_liquid_valve
    Textfield (780,753 78x25), "%1.2f bar", text variable: Chiller_3.Oil_Filter_Drop
        p4168582468: Chiller_3.Oil_Filter_Drop
    Label (778,732 83x22), "Oil filter drop"
    Textfield (667,814 92x25), "%1.0f %%", text variable: Chiller_3.Liquid_valve_output
        p4168582468: Chiller_3.Liquid_valve_output
    Label (646,788 135x30), "Liquid valve order"
    Textfield (780,703 78x25), "%1.2f bar", text variable: Chiller_3.Press_oil_receiver
        p4168582468: Chiller_3.Press_oil_receiver
    Label (752,682 135x22), "Oil pressure receiver"
    Textfield (780,654 78x25), "%1.1f °C", text variable: Chiller_3.Oil_temp_receiver
        p4168582468: Chiller_3.Oil_temp_receiver
    Label (748,633 143x22), "Oil temperature receiver"
    Textfield (780,605 78x25), "%1.2f bar", text variable: Chiller_3.Oil_diff_pressure
        p4168582468: Chiller_3.Oil_diff_pressure
    Label (769,584 101x22), "Oil diff pressure"
    Label (736,136 109x24), "Prerotary position"
    Textfield (754,159 72x25), "%1.0f %%", text variable: Chiller_3.Feedback_PRV
        p4168582468: Chiller_3.Feedback_PRV
    Label (746,83 87x24), "VGD position"
    Textfield (753,106 72x25), "%1.0f %%", text variable: Chiller_3.Feedback_VGD
        p4168582468: Chiller_3.Feedback_VGD
    Label (746,31 87x24), "Stall detector"
    Textfield (753,54 72x25), "%1.2f V", text variable: Chiller_3.Stall_detector
        p4168582468: Chiller_3.Stall_detector
    Label (1067,211 171x24), "Suction pressure saturated"
    Textfield (1116,234 72x25), "%1.1f °C", text variable: Chiller_3.Suction_saturated_temp
        p4168582468: Chiller_3.Suction_saturated_temp
    Textfield (1116,291 72x25), "%1.1f bara", text variable: Chiller_3.Press_suction_compr
        p4168582468: Chiller_3.Press_suction_compr
    Label (1067,268 171x24), "Suction pressure"
    Textfield (1116,368 72x25), "%1.1f °C", text variable: Chiller_3.Theta_out
        p4168582468: Chiller_3.Theta_out
    Label (1111,345 83x24), "Theta out"
    Label (1196,557 84x27), "CW pressure"
    Textfield (1200,581 77x25), "%1.2f bar", text variable: Chiller_3.Press_chilled_medium_out
        p4168582468: Chiller_3.Press_chilled_medium_out
    Textfield (1200,710 77x25), "%1.2f bar", text variable: Chiller_3.Press_chilled_medium_in
        p4168582468: Chiller_3.Press_chilled_medium_in
    Label (1196,686 84x27), "CW pressure"
    Textfield (1170,506 72x25), "%1.1f °C", text variable: Chiller_3.Temp_chilled_medium_out
        p4168582468: Chiller_3.Temp_chilled_medium_out
    Label (1146,483 121x24), "Chilled water outlet"
    Label (1146,428 121x24), "CW setpoint"
    Textfield (1170,451 72x25), "%1.1f °C", text variable: Chiller_3.SP_CW_controller
        p4168582468: Chiller_3.SP_CW_controller
    Label (1252,619 84x30), "Diff pressure"
    Textfield (1256,648 77x25), "%1.2f bar", text variable: Chiller_3.dP_CW
        p4168582468: Chiller_3.dP_CW
    Textfield (1170,783 72x25), "%1.1f °C", text variable: Chiller_3.Temp_chilled_medium_in
        p4168582468: Chiller_3.Temp_chilled_medium_in
    Label (1146,760 121x24), "Chilled water inlet"
    Group (6,271 190x25)
        Rectangle (0,0 190x25)
        Label (0,2 105x21), "Running"
        Lamp1 (166,3 23x20), variable: Chiller_3.Unit_running, style: Lamp-Lamp1-Green
    Group (6,163 190x25)
        Rectangle (0,0 190x25)
        Label (1,2 105x21), "Auto"
        Lamp1 (166,3 23x20), variable: Chiller_3.Unit_auto, style: Lamp-Lamp1-Green
    Group (6,199 190x25)
        Rectangle (0,0 190x25)
        Label (0,2 105x21), "Remote"
        Lamp1 (166,3 23x20), variable: Chiller_3.Unit_remote, style: Lamp-Lamp1-Green
    Group (6,235 190x25)
        Rectangle (0,0 190x25)
        Label (0,2 105x21), "Manual"
        Lamp1 (166,3 23x20), variable: Chiller_3.Unit_manual, style: Lamp-Lamp1-Green
    Group (6,307 190x25)
        Rectangle (0,0 190x25)
        Label (1,2 105x21), "Available"
        Lamp1 (166,3 23x20), variable: Chiller_3.Unit_available, style: Lamp-Lamp1-Green
    Group (6,343 190x25)
        Rectangle (0,0 190x25)
        Label (0,2 130x21), "Start switch"
        Lamp1 (166,3 23x20), variable: Chiller_3.Unit_start_switch, style: Lamp-Lamp1-Green
    Group (6,381 190x25)
        Rectangle (0,0 190x25)
        Label (0,2 160x21), "Comms sequence"
        Lamp1 (166,3 23x20), variable: not.Sequence.A_Comms_Chiller_3, style: Lamp-Lamp1-Green
    Label (912,265 95x24), "Oil temp comp."
    Textfield (923,288 72x25), "%1.1f °C", text variable: Chiller_3.Temp_oil_inlet_compr
        p4168582468: Chiller_3.Temp_oil_inlet_compr
    Label (902,324 115x24), "Oil pressure [HP]"
    Textfield (923,347 72x25), "%1.2f bar", text variable: Chiller_3.Press_oil_compr
        p4168582468: Chiller_3.Press_oil_compr
    Image (921,41 317x130), invisible if: Chiller_3.Unit_alarm, image: ImagePool.ALARM
    Image (921,41 317x130), invisible if: Chiller_3.Unit_trip, image: ImagePool.TRIP
    Label (7,87 89x30), "Mode"
    Label (106,87 89x30), "Status"
    Rectangle (334,160 48x246)
    Image (238,160 48x246), image: ImagePool.CapBarTranparant
    BarDisplayImage (239,161 46x242), value: Sequence.Seq_cap_order_C3, style: BarDisplayImage-Gray, scale format: %.0f, scale 0..100
        p3451962224: ImagePool.Invisible
    Rectangle (673,210 36x36), colour toggle: Chiller_3.Unit_running
    Rectangle (673,210 36x36), colour toggle: Chiller_3.Unit_alarm
    Rectangle (673,210 36x36), colour toggle: Chiller_3.Unit_trip
    Image (334,160 48x246), image: ImagePool.CapBarTranparant
    BarDisplayImage (335,161 46x242), value: Chiller_3.Chiller_capacity_t1, style: BarDisplayImage-Gray, scale format: %.0f, scale 0..100
        p3451962224: ImagePool.Invisible
    Rectangle (493,624 28x52)
    Image (493,624 29x54), image: ImagePool.CapBarTranparant
    BarDisplayImage (494,625 27x51), value: Chiller_3.Liquid_level_condenser, style: BarDisplayImage-Gray, scale format: %.0f, scale 0..100
        p3451962224: ImagePool.Invisible
    Image (95,742 147x16), image: ImagePool.PipeGreen_1_Horizontal
    Textfield (605,753 92x25), "%1.1f °C", text variable: Chiller_3.Liquid_line_temp
        p4168582468: Chiller_3.Liquid_line_temp
    Label (595,727 113x30), "Liquid line temp"
    Image (228,490 57x88), image: ImagePool.Valve_3
    Label (115,461 105x30), "Sea water valve order"
    Textfield (129,492 76x25), "%1.0f %%", text variable: Chiller_3.Order_SWW_overboard
        p4168582468: Chiller_3.Order_SWW_overboard
    Label (281,461 105x30), "Sea water valve pos"
    Textfield (295,492 76x25), "%1.0f %%", text variable: Chiller_3.Feedback_seawater_valve_overboard
        p4168582468: Chiller_3.Feedback_seawater_valve_overboard
    Group (37,610 180x72)
        Rectangle (0,0 180x72)
        Label (0,0 180x72), "Sea water valve Pos. 100% = Max. overboard Pos. 0% = Max. recirculation"
    Label (511,138 103x22), "Temp winding"
    Rectangle (1274,37 207x30)
    Label (1310,38 142x28), "Time between starts"
    Lamp1 (1281,43 23x20), variable: Chiller_3.Start_inhib_time_between_Start, style: Lamp-Lamp1-Green
    Rectangle (1274,67 207x30)
    Label (1310,68 162x28), "Time between stop / starts"
    Lamp1 (1281,73 23x20), variable: Chiller_3.Start_inhib_time_between_Stop_Start, style: Lamp-Lamp1-Green
    Label (1307,7 140x24), "Start inhibits"
    Rectangle (1274,97 207x30)
    Label (1310,98 162x28), "Cold oil in oil receiver"
    Lamp1 (1281,103 23x20), variable: Chiller_3.Start_inhib_time_Oil_receiver_temp, style: Lamp-Lamp1-Green
    Rectangle (1274,127 207x30)
    Label (1310,128 162x28), "PRV not in min position"
    Lamp1 (1281,133 23x20), variable: Chiller_3.Start_inhib_PRV_not_min, style: Lamp-Lamp1-Green
    Rectangle (1274,157 207x30)
    Label (1310,158 162x28), "Main braker inserted"
    Lamp1 (1281,163 23x20), variable: not.Chiller_3.DO_9_0_Main_breaker_ready, style: Lamp-Lamp1-Green
    Rectangle (1274,187 207x30)
    Label (1310,188 162x28), "Motor overload protection"
    Lamp1 (1281,193 23x20), variable: not.Chiller_3.DI_0_6_Overload_protection, style: Lamp-Lamp1-Green
END_VISUALIZATION

// /Chiller_3_Oil
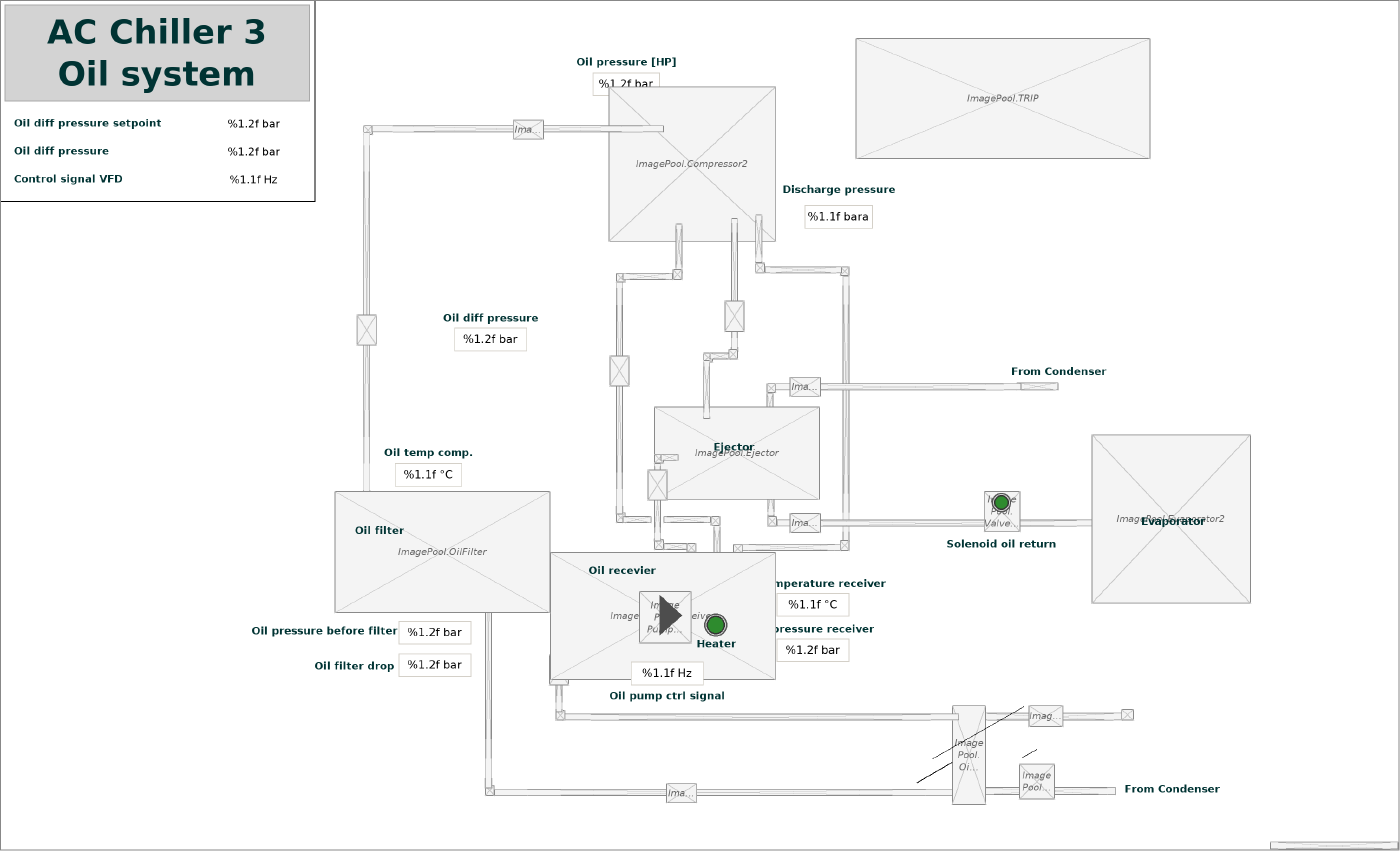
VISUALIZATION Chiller_3_Oil  // 1507x917
    Image (1094,412 45x8), angle 180, image: ImagePool.PipeBlack_1S_H_Faded
    Rectangle (0,0 339x217)
    Image (1367,907 138x8), angle 270, image: ImagePool.PipeGrey_1S_Horizontal
    Image (1053,768 155x8), image: ImagePool.PipeGrey_1S_Horizontal
    Image (1207,764 13x12), image: ImagePool.PipeGrey_3_LU
    Textfield (5,5 328x104), "AC Chiller 3 Oil system"
    Label (1066,387 128x27), "From Condenser"
    Label (838,191 129x27), "Discharge pressure"
    Textfield (866,221 73x25), "%1.1f bara", text variable: Chiller_3.Press_discharge_compr
        p4168582468: Chiller_3.Press_discharge_compr
    Label (1007,573 142x27), "Solenoid oil return"
    Textfield (429,704 78x25), "%1.2f bar", text variable: Chiller_3.Oil_Filter_Drop
        p4168582468: Chiller_3.Oil_Filter_Drop
    Label (340,707 83x22), "Oil filter drop"
    Textfield (836,688 78x25), "%1.2f bar", text variable: Chiller_3.Press_oil_receiver
        p4168582468: Chiller_3.Press_oil_receiver
    Label (808,667 135x22), "Oil pressure receiver"
    Textfield (836,639 78x25), "%1.1f °C", text variable: Chiller_3.Oil_temp_receiver
        p4168582468: Chiller_3.Oil_temp_receiver
    Label (804,618 143x22), "Oil temperature receiver"
    Textfield (489,353 78x25), "%1.2f bar", text variable: Chiller_3.Oil_diff_pressure
        p4168582468: Chiller_3.Oil_diff_pressure
    Label (478,332 101x22), "Oil diff pressure"
    Label (414,476 95x24), "Oil temp comp."
    Textfield (425,499 72x25), "%1.1f °C", text variable: Chiller_3.Temp_oil_inlet_compr
        p4168582468: Chiller_3.Temp_oil_inlet_compr
    Label (617,55 115x24), "Oil pressure [HP]"
    Textfield (638,78 72x25), "%1.2f bar", text variable: Chiller_3.Press_oil_compr
        p4168582468: Chiller_3.Press_oil_compr
    Image (921,41 317x130), invisible if: Chiller_3.Unit_alarm, image: ImagePool.ALARM
    Image (921,41 317x130), invisible if: Chiller_3.Unit_trip, image: ImagePool.TRIP
    Textfield (238,122 70x23), "%1.2f bar", text variable: Chiller_3.SP_oil_pressure
    Label (12,118 193x30), "Oil diff pressure setpoint"
    Textfield (238,152 70x23), "%1.2f bar", text variable: Chiller_3.Oil_diff_pressure
    Label (12,148 193x30), "Oil diff pressure"
    Textfield (238,182 70x23), "%1.1f Hz", text variable: Chiller_3.Setpoint_conv_oil_pump
    Label (12,178 131x30), "Control signal VFD"
    Label (651,739 135x22), "Oil pump ctrl signal"
    Textfield (429,669 78x25), "%1.2f bar", text variable: Chiller_3.Oil_pressure_before_filter
        p4168582468: Chiller_3.Oil_pressure_before_filter
    Label (276,669 147x22), "Oil pressure before filter"
    Label (1210,837 106x27), "From Condenser"
    Image (655,93 180x167), image: ImagePool.Compressor2
    Image (1051,848 150x8), angle 180, image: ImagePool.PipeBlack_1S_H_Faded
    Image (798,586 108x7), image: ImagePool.PipeBlack_1_Horizontal
    Image (907,297 7x286), image: ImagePool.PipeBlack_1_Vertical
    Image (391,135 10x10), image: ImagePool.PipeBlack_1_RD
    Image (522,846 10x11), image: ImagePool.PipeBlack_1_RU
    Image (1107,760 37x23), image: ImagePool.Arrow gray right
    Image (836,560 348x7), image: ImagePool.PipeBlack_1_Horizontal
    Image (1175,468 171x182), image: ImagePool.Evaporator2
    Image (826,512 7x44), image: ImagePool.PipeBlack_1_Vertical
    Image (826,556 10x11), image: ImagePool.PipeBlack_1_RU
    Image (789,596 7x28), image: ImagePool.PipeBlack_1_Vertical
    Image (789,586 10x10), image: ImagePool.PipeBlack_1_RD
    Image (904,582 10x11), image: ImagePool.PipeBlack_1_LU
    Image (850,553 33x21), image: ImagePool.Arrow black left
    Image (904,287 10x10), image: ImagePool.PipeBlack_1_LD
    Image (823,287 83x7), image: ImagePool.PipeBlack_1_Horizontal
    Image (813,283 10x11), image: ImagePool.PipeBlack_1_RU
    Image (813,231 7x52), image: ImagePool.PipeBlack_1_Vertical
    Image (825,413 10x10), image: ImagePool.PipeBlack_1_RD
    Image (834,413 265x7), image: ImagePool.PipeBlack_1_Horizontal
    Image (825,423 7x28), image: ImagePool.PipeBlack_1_Vertical
    Image (704,438 178x100), image: ImagePool.Ejector
    Image (850,406 33x21), image: ImagePool.Arrow black left
    Image (532,850 500x7), image: ImagePool.PipeBlack_1_Horizontal
    Image (1025,760 36x107), image: ImagePool.OilHeatExchanger
    Image (605,769 427x7), image: ImagePool.PipeBlack_1_Horizontal
    Image (598,765 10x11), image: ImagePool.PipeBlack_1_RU
    Image (598,670 7x97), image: ImagePool.PipeBlack_1_Vertical
    Image (598,660 10x10), image: ImagePool.PipeBlack_1_RD
    Image (605,660 19x7), image: ImagePool.PipeBlack_1_Horizontal
    Image (591,705 21x33), image: ImagePool.Arrow black down
    Image (717,844 33x21), image: ImagePool.Arrow black left
    Image (768,566 7x50), image: ImagePool.PipeBlack_1_Vertical
    Image (765,556 10x10), image: ImagePool.PipeBlack_1_LD
    Image (714,556 51x7), image: ImagePool.PipeBlack_1_Horizontal
    Image (704,581 10x11), image: ImagePool.PipeBlack_1_RU
    Image (704,499 7x84), image: ImagePool.PipeBlack_1_Vertical
    Image (704,489 10x10), image: ImagePool.PipeBlack_1_RD
    Image (711,489 19x7), image: ImagePool.PipeBlack_1_Horizontal
    Image (697,506 21x33), image: ImagePool.Arrow black down
    Image (714,585 28x7), image: ImagePool.PipeBlack_1_Horizontal
    Image (739,585 10x10), image: ImagePool.PipeBlack_1_LD
    Image (742,595 7x21), image: ImagePool.PipeBlack_1_Vertical
    Image (592,595 243x137), image: ImagePool.OilReceiver
    Image (400,135 314x7), image: ImagePool.PipeBlack_1_Horizontal
    Label (630,604 80x22), "Oil recevier"
    Image (522,553 7x296), image: ImagePool.PipeBlack_1_Vertical
    Image (519,544 10x10), image: ImagePool.PipeBlack_1_LD
    Image (400,544 120x7), image: ImagePool.PipeBlack_1_Horizontal
    Image (391,540 10x11), image: ImagePool.PipeBlack_1_RU
    Image (391,142 7x400), image: ImagePool.PipeBlack_1_Vertical
    Image (663,552 10x11), image: ImagePool.PipeBlack_1_RU
    Image (663,301 7x253), image: ImagePool.PipeBlack_1_Vertical
    Image (663,294 10x10), image: ImagePool.PipeBlack_1_RD
    Image (670,294 54x7), image: ImagePool.PipeBlack_1_Horizontal
    Image (656,383 21x33), image: ImagePool.Arrow black down
    Image (670,556 31x7), image: ImagePool.PipeBlack_1_Horizontal
    Image (727,241 7x53), image: ImagePool.PipeBlack_1_Vertical
    Image (724,290 10x11), image: ImagePool.PipeBlack_1_LU
    Image (757,380 10x10), image: ImagePool.PipeBlack_1_RD
    Image (764,380 22x7), image: ImagePool.PipeBlack_1_Horizontal
    Image (787,235 7x144), image: ImagePool.PipeBlack_1_Vertical
    Image (784,376 10x11), image: ImagePool.PipeBlack_1_LU
    Image (757,388 7x63), image: ImagePool.PipeBlack_1_Vertical
    Image (780,324 21x33), image: ImagePool.Arrow black down
    Label (750,471 80x22), "Ejector"
    Label (1223,551 80x22), "Evaporator"
    Image (384,339 21x33), image: ImagePool.Arrow black up
    Image (552,129 33x21), image: ImagePool.Arrow black right
    Image (360,529 232x131), image: ImagePool.OilFilter
    Label (379,561 59x22), "Oil filter"
    Line (987,843) (1025,821)
    Line (1100,816) (1116,807)
    Line (1004,817) (1102,761)
    Image (1097,823 38x38), image: ImagePool.RegValve
    Image (688,637 56x56), image: ImagePool.Pump_Large_3
    Polygon (710,660) (710,641) (734,663) (710,684) (710,676), colour toggle: Chiller_3.Comp_oil_pump
    Lamp1 (756,656 29x35), variable: Chiller_3.DO_0_6_Oil_heater, style: Lamp-Lamp1-Green
    Label (744,683 55x22), "Heater"
    Image (1059,529 39x44), image: ImagePool.Valve_2
    Lamp1 (1066,529 24x25), variable: Chiller_3.DO_0_4_Solenoid_valve_oil, style: Lamp-Lamp1-Green
    Textfield (679,713 78x25), "%1.1f Hz", text variable: Chiller_3.Setpoint_conv_oil_pump
END_VISUALIZATION

// /Homepage
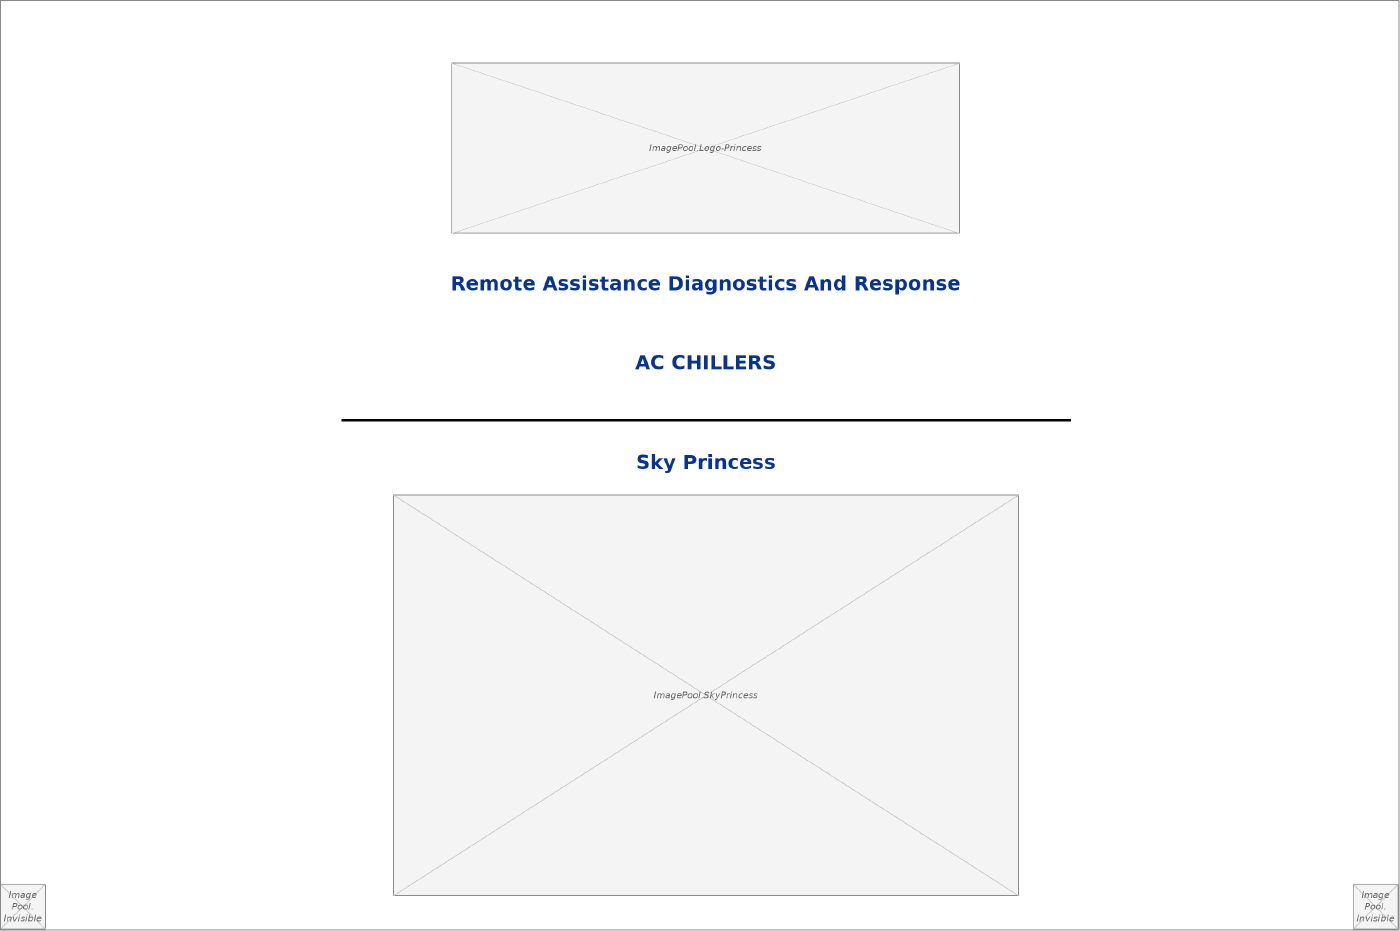
VISUALIZATION Homepage  // 1542x1026
    Label (490,287 575x51), "Remote Assistance Diagnostics And Response"
    Label (597,484 361x51), "Sky Princess"
    Rectangle (376,462 803x2)
    Label (597,374 361x51), "AC CHILLERS"
    Image (0,974 50x50), image: ImagePool.Invisible
    Image (1490,974 50x50), image: ImagePool.Invisible
    Image (433,545 689x442), image: ImagePool.SkyPrincess
    Image (497,69 560x188), image: ImagePool.Logo-Princess
END_VISUALIZATION

(* text list Chiller_trendvalues (id | default)
  0 | Clear values
  1 | Chiller Capacity t1
  2 | Control Signal SW Valve
  3 | dP CW
  4 | dP SW
  5 | Feedback Hot Gas Valve
  6 | Feedback Liquid Valve
  7 | Feedback PRV
  8 | Feedback Sea Water Valve
  9 | Feedback VGD
  10 | Hot Gas Valve Order
  11 | Liquid Level Condenser
  12 | Liquid Valve Order
  13 | Motor Current
  14 | Pressure CW Inlet
  15 | Pressure CW Outlet
  16 | Pressure Oil Compressor
  17 | Pressure Oil Diff
  18 | Pressure Oil Receiver
  19 | Pressure Suction Saturated
  20 | Pressure SW Inlet
  21 | Pressure SW Outlet
  22 | Sea Water Valve Order
  23 | Setpoint Liquid Level
  24 | Temp Chilled Medium Inlet
  25 | Temp Chilled Medium Outlet
  26 | Temp Discharge Gas
  27 | Temp Discharge Saturated
  28 | Temp Discharge Superheat
  29 | Temp Motor Air
  30 | Temp Motor Bearing DE
  31 | Temp Motor Bearing NDE
  32 | Temp Motor Winding R
  33 | Temp Motor Winding S
  34 | Temp Motor Winding T
  35 | Temp Oil Inlet Compressor
  36 | Temp Sea Water Inlet
  37 | Temp Suction Saturated
  38 | Theta Out
  39 | Thrust Bearing position
   |  *)

(* text list Chiller_VSD_trendvalues (id | default)
  0 | Clear values
  1 | Chiller Capacity t1
  2 | Control Signal SW Valve
  3 | dP CW
  4 | dP SW
  5 | Feedback Hot Gas Valve
  6 | Feedback Liquid Valve
  7 | Feedback PRV
  8 | Feedback Sea Water Valve
  9 | Feedback VGD
  10 | Hot Gas Valve Order
  11 | Liquid Level Condenser
  12 | Liquid Valve Order
  13 | Motor Current
  14 | Pressure CW Inlet
  15 | Pressure CW Outlet
  16 | Pressure Oil Compressor
  17 | Pressure Oil Diff
  18 | Pressure Oil Receiver
  19 | Pressure Suction Saturated
  20 | Pressure SW Inlet
  21 | Pressure SW Outlet
  22 | Sea Water Valve Order
  23 | Setpoint Liquid Level
  24 | Temp Chilled Medium Inlet
  25 | Temp Chilled Medium Outlet
  26 | Temp Discharge Gas
  27 | Temp Discharge Saturated
  28 | Temp Discharge Superheat
  29 | Temp Motor Air
  30 | Temp Motor Bearing DE
  31 | Temp Motor Bearing NDE
  32 | Temp Motor Winding R
  33 | Temp Motor Winding S
  34 | Temp Motor Winding T
  35 | Temp Oil Inlet Compressor
  36 | Temp Sea Water Inlet
  37 | Temp Suction Saturated
  38 | Theta Out
  39 | Thrust Bearing position
  40 | VFD Current Speed Hz
  41 | VFD Order Hz
   |  *)

(* text list TextList_Local_IAMCS (id | default)
  0 | Local
  1 | IAMCS
   |  *)
